LIN {X 0,Y 469.971,Z 691.931,A -85,B 0,C 180,E1 20930.891,E2 20930.891} C_VEL
LIN {X 0,Y 471.709,Z 664.852,A -85,B 0,C 180,E1 20927.125,E2 20927.125} C_VEL
LIN {X 0,Y 473.117,Z 644.354,A -85,B 0,C 180,E1 20924.22,E2 20924.22} C_VEL
LIN {X 0,Y 468.98,Z 629.083,A -85,B 0,C 180,E1 20921.533,E2 20921.533} C_VEL
LIN {X 0,Y 465.017,Z 616.426,A -85,B 0,C 180,E1 20919.107,E2 20919.107} C_VEL
LIN {X 0,Y 465.008,Z 616.312,A -85,B 0,C 180,E1 20915.42,E2 20915.42} C_VEL
LIN {X 0,Y 465.004,Z 616.306,A -85,B 0,C 180,E1 20911.79,E2 20911.79} C_VEL
LIN {X 0,Y 465.007,Z 616.308,A -85,B 0,C 180,E1 20908.093,E2 20908.093} C_VEL
LIN {X 0,Y 465.007,Z 616.309,A -85,B 0,C 180,E1 20904.384,E2 20904.384} C_VEL
LIN {X 0,Y 465.007,Z 616.309,A -85,B 0,C 180,E1 20900.649,E2 20900.649} C_VEL
LIN {X 0,Y 465.005,Z 616.31,A -85,B 0,C 180,E1 20897.004,E2 20897.004} C_VEL
LIN {X 0,Y 465,Z 616.311,A -85,B 0,C 180,E1 20893.302,E2 20893.302} C_VEL
LIN {X 0,Y 465.008,Z 616.3,A -85,B 0,C 180,E1 20889.655,E2 20889.655} C_VEL
LIN {X 0,Y 465.009,Z 616.303,A -85,B 0,C 180,E1 20886.048,E2 20886.048} C_VEL
LIN {X 0,Y 465.002,Z 616.308,A -85,B 0,C 180,E1 20882.342,E2 20882.342} C_VEL
LIN {X 0,Y 464.997,Z 616.312,A -85,B 0,C 180,E1 20878.645,E2 20878.645} C_VEL
LIN {X 0,Y 465.008,Z 616.299,A -85,B 0,C 180,E1 20874.943,E2 20874.943} C_VEL
LIN {X 0,Y 465.01,Z 616.3,A -85,B 0,C 180,E1 20871.344,E2 20871.344} C_VEL
LIN {X 0,Y 465,Z 616.307,A -85,B 0,C 180,E1 20867.709,E2 20867.709} C_VEL
LIN {X 0,Y 464.992,Z 616.314,A -85,B 0,C 180,E1 20864.024,E2 20864.024} C_VEL
LIN {X 0,Y 465.01,Z 616.302,A -85,B 0,C 180,E1 20860.353,E2 20860.353} C_VEL
LIN {X 0,Y 465.01,Z 616.299,A -85,B 0,C 180,E1 20856.654,E2 20856.654} C_VEL
LIN {X 0,Y 465,Z 616.302,A -85,B 0,C 180,E1 20853.019,E2 20853.019} C_VEL
LIN {X 0,Y 464.988,Z 616.304,A -85,B 0,C 180,E1 20849.362,E2 20849.362} C_VEL
LIN {X 0,Y 465.009,Z 616.305,A -85,B 0,C 180,E1 20845.712,E2 20845.712} C_VEL
LIN {X 0,Y 465.014,Z 616.304,A -85,B 0,C 180,E1 20842.052,E2 20842.052} C_VEL
LIN {X 0,Y 464.994,Z 616.31,A -85,B 0,C 180,E1 20838.442,E2 20838.442} C_VEL
LIN {X 0,Y 464.987,Z 616.314,A -85,B 0,C 180,E1 20834.798,E2 20834.798} C_VEL
LIN {X 0,Y 465.018,Z 616.309,A -85,B 0,C 180,E1 20831.143,E2 20831.143} C_VEL
LIN {X 0,Y 465.05,Z 616.559,A -85,B 0,C 180,E1 20829.524,E2 20829.524} C_VEL
LIN {X 0,Y 470.586,Z 631.403,A -85,B 0,C 180,E1 20827.379,E2 20827.379} C_VEL
LIN {X 0,Y 477.306,Z 651.198,A -85,B 0,C 180,E1 20824.859,E2 20824.859} C_VEL
LIN {X 0,Y 474.522,Z 692.791,A -85,B 0,C 180,E1 20821.157,E2 20821.157} C_VEL
LIN {X 0,Y 473.708,Z 708.918,A -85,B 0,C 180,E1 20819.787,E2 20819.787} C_VEL
LIN {X 0,Y 476.659,Z 731.259,A -85,B 0,C 180,E1 20819.245,E2 20819.245} C_VEL
LIN {X 0,Y 474.227,Z 923.8,A -85,B 0,C 180,E1 20816.242,E2 20816.242} C_VEL
LIN {X 0,Y 473.509,Z 943.256,A -85,B 0,C 180,E1 20815.721,E2 20815.721} C_VEL
LIN {X 0,Y 472.588,Z 962.087,A -85,B 0,C 180,E1 20814.99,E2 20814.99} C_VEL
LIN {X 0,Y 471.547,Z 979.642,A -85,B 0,C 180,E1 20814.09,E2 20814.09} C_VEL
LIN {X 0,Y 470.395,Z 997.145,A -85,B 0,C 180,E1 20812.957,E2 20812.957} C_VEL
LIN {X 0,Y 469.201,Z 1013.781,A -85,B 0,C 180,E1 20811.633,E2 20811.633} C_VEL
LIN {X 0,Y 468.041,Z 1029.511,A -85,B 0,C 180,E1 20810.117,E2 20810.117} C_VEL
LIN {X 0,Y 466.991,Z 1043.8,A -85,B 0,C 180,E1 20808.47,E2 20808.47} C_VEL
LIN {X 0,Y 466.038,Z 1057.494,A -85,B 0,C 180,E1 20806.579,E2 20806.579} C_VEL
LIN {X 0,Y 465.315,Z 1068.946,A -85,B 0,C 180,E1 20804.688,E2 20804.688} C_VEL
LIN {X 0,Y 464.744,Z 1079.076,A -85,B 0,C 180,E1 20802.676,E2 20802.676} C_VEL
LIN {X 0,Y 464.358,Z 1087.812,A -85,B 0,C 180,E1 20800.546,E2 20800.546} C_VEL
LIN {X 0,Y 464.099,Z 1095.056,A -85,B 0,C 180,E1 20798.299,E2 20798.299} C_VEL
LIN {X 0,Y 463.962,Z 1100.677,A -85,B 0,C 180,E1 20795.937,E2 20795.937} C_VEL
LIN {X 0,Y 463.915,Z 1104.2,A -85,B 0,C 180,E1 20793.707,E2 20793.707} C_VEL
LIN {X 0,Y 463.911,Z 1106.031,A -85,B 0,C 180,E1 20791.482,E2 20791.482} C_VEL
LIN {X 0,Y 463.912,Z 1106.28,A -85,B 0,C 180,E1 20789.259,E2 20789.259} C_VEL
LIN {X 0,Y 463.911,Z 1104.962,A -85,B 0,C 180,E1 20787.035,E2 20787.035} C_VEL
LIN {X 0,Y 463.937,Z 1102.003,A -85,B 0,C 180,E1 20784.806,E2 20784.806} C_VEL
LIN {X 0,Y 464.031,Z 1097.327,A -85,B 0,C 180,E1 20782.571,E2 20782.571} C_VEL
LIN {X 0,Y 464.235,Z 1090.845,A -85,B 0,C 180,E1 20780.328,E2 20780.328} C_VEL
LIN {X 0,Y 464.56,Z 1082.932,A -85,B 0,C 180,E1 20778.201,E2 20778.201} C_VEL
LIN {X 0,Y 465.072,Z 1073.039,A -85,B 0,C 180,E1 20776.067,E2 20776.067} C_VEL
LIN {X 0,Y 465.772,Z 1061.653,A -85,B 0,C 180,E1 20774.051,E2 20774.051} C_VEL
LIN {X 0,Y 466.645,Z 1048.784,A -85,B 0,C 180,E1 20772.157,E2 20772.157} C_VEL
LIN {X 0,Y 467.708,Z 1034.369,A -85,B 0,C 180,E1 20770.389,E2 20770.389} C_VEL
LIN {X 0,Y 468.856,Z 1018.933,A -85,B 0,C 180,E1 20768.809,E2 20768.809} C_VEL
LIN {X 0,Y 470.058,Z 1002.565,A -85,B 0,C 180,E1 20767.422,E2 20767.422} C_VEL
LIN {X 0,Y 471.25,Z 985.312,A -85,B 0,C 180,E1 20766.226,E2 20766.226} C_VEL
LIN {X 0,Y 472.364,Z 967.12,A -85,B 0,C 180,E1 20765.221,E2 20765.221} C_VEL
LIN {X 0,Y 473.338,Z 948.404,A -85,B 0,C 180,E1 20764.433,E2 20764.433} C_VEL
LIN {X 0,Y 474.13,Z 929.225,A -85,B 0,C 180,E1 20763.861,E2 20763.861} C_VEL
LIN {X 0,Y 474.605,Z 906.118,A -85,B 0,C 180,E1 20763.436,E2 20763.436} C_VEL
LIN {X 0,Y 476.595,Z 728.668,A -85,B 0,C 180,E1 20760.68,E2 20760.68} C_VEL
LIN {X 0,Y 473.739,Z 708.363,A -85,B 0,C 180,E1 20760.163,E2 20760.163} C_VEL
LIN {X 0,Y 476.269,Z 665.707,A -85,B 0,C 180,E1 20756.454,E2 20756.454} C_VEL
LIN {X 0,Y 477.119,Z 650.714,A -85,B 0,C 180,E1 20755.103,E2 20755.103} C_VEL
LIN {X 0,Y 469.453,Z 628.767,A -85,B 0,C 180,E1 20752.401,E2 20752.401} C_VEL
LIN {X 0,Y 465.04,Z 616.516,A -85,B 0,C 180,E1 20750.749,E2 20750.749} C_VEL
LIN {X 0,Y 465.004,Z 616.313,A -85,B 0,C 180,E1 20747.157,E2 20747.157} C_VEL
LIN {X 0,Y 465,Z 616.308,A -85,B 0,C 180,E1 20743.478,E2 20743.478} C_VEL
LIN {X 0,Y 465.016,Z 616.309,A -85,B 0,C 180,E1 20739.847,E2 20739.847} C_VEL
LIN {X 0,Y 464.999,Z 616.313,A -85,B 0,C 180,E1 20736.25,E2 20736.25} C_VEL
LIN {X 0,Y 465.008,Z 616.313,A -85,B 0,C 180,E1 20732.517,E2 20732.517} C_VEL
LIN {X 0,Y 465.014,Z 616.311,A -85,B 0,C 180,E1 20728.792,E2 20728.792} C_VEL
LIN {X 0,Y 465.012,Z 616.31,A -85,B 0,C 180,E1 20725.061,E2 20725.061} C_VEL
LIN {X 0,Y 464.987,Z 616.312,A -85,B 0,C 180,E1 20721.395,E2 20721.395} C_VEL
LIN {X 0,Y 464.98,Z 616.317,A -85,B 0,C 180,E1 20717.649,E2 20717.649} C_VEL
LIN {X 0,Y 465.006,Z 616.315,A -85,B 0,C 180,E1 20714.062,E2 20714.062} C_VEL
LIN {X 0,Y 465.01,Z 616.312,A -85,B 0,C 180,E1 20710.405,E2 20710.405} C_VEL
LIN {X 0,Y 465.002,Z 616.567,A -85,B 0,C 180,E1 20709.311,E2 20709.311} C_VEL
LIN {X 0,Y 469.677,Z 632.432,A -85,B 0,C 180,E1 20707.215,E2 20707.215} C_VEL
LIN {X 0,Y 471.206,Z 640.102,A -85,B 0,C 180,E1 20706.274,E2 20706.274} C_VEL
LIN {X 0,Y 471.027,Z 671.519,A -85,B 0,C 180,E1 20702.737,E2 20702.737} C_VEL
LIN {X 0,Y 470.651,Z 698.884,A -85,B 0,C 180,E1 20699.574,E2 20699.574} C_VEL
LIN {X 0,Y 470.561,Z 708.868,A -85,B 0,C 180,E1 20698.432,E2 20698.432} C_VEL
LIN {X 0,Y 471.035,Z 713.013,A -85,B 0,C 180,E1 20698.329,E2 20698.329} C_VEL
LIN {X 0,Y 469.379,Z 847.569,A -85,B 0,C 180,E1 20696.041,E2 20696.041} C_VEL
LIN {X 0,Y 469.234,Z 863.454,A -85,B 0,C 180,E1 20695.554,E2 20695.554} C_VEL
LIN {X 0,Y 468.89,Z 879.333,A -85,B 0,C 180,E1 20694.826,E2 20694.826} C_VEL
LIN {X 0,Y 468.431,Z 893.617,A -85,B 0,C 180,E1 20693.935,E2 20693.935} C_VEL
LIN {X 0,Y 467.831,Z 908.134,A -85,B 0,C 180,E1 20692.756,E2 20692.756} C_VEL
LIN {X 0,Y 467.229,Z 920.197,A -85,B 0,C 180,E1 20691.508,E2 20691.508} C_VEL
LIN {X 0,Y 466.592,Z 931.837,A -85,B 0,C 180,E1 20690.004,E2 20690.004} C_VEL
LIN {X 0,Y 466.055,Z 941.162,A -85,B 0,C 180,E1 20688.491,E2 20688.491} C_VEL
LIN {X 0,Y 465.573,Z 949.787,A -85,B 0,C 180,E1 20686.715,E2 20686.715} C_VEL
LIN {X 0,Y 465.223,Z 956.426,A -85,B 0,C 180,E1 20684.926,E2 20684.926} C_VEL
LIN {X 0,Y 464.953,Z 961.615,A -85,B 0,C 180,E1 20682.994,E2 20682.994} C_VEL
LIN {X 0,Y 464.788,Z 965.016,A -85,B 0,C 180,E1 20681.044,E2 20681.044} C_VEL
LIN {X 0,Y 464.699,Z 966.73,A -85,B 0,C 180,E1 20678.941,E2 20678.941} C_VEL
LIN {X 0,Y 464.68,Z 966.571,A -85,B 0,C 180,E1 20676.945,E2 20676.945} C_VEL
LIN {X 0,Y 464.716,Z 964.62,A -85,B 0,C 180,E1 20674.921,E2 20674.921} C_VEL
LIN {X 0,Y 464.835,Z 960.927,A -85,B 0,C 180,E1 20672.939,E2 20672.939} C_VEL
LIN {X 0,Y 465.064,Z 955.222,A -85,B 0,C 180,E1 20670.929,E2 20670.929} C_VEL
LIN {X 0,Y 465.382,Z 948.093,A -85,B 0,C 180,E1 20669.103,E2 20669.103} C_VEL
LIN {X 0,Y 465.852,Z 938.867,A -85,B 0,C 180,E1 20667.284,E2 20667.284} C_VEL
LIN {X 0,Y 466.395,Z 928.44,A -85,B 0,C 180,E1 20665.679,E2 20665.679} C_VEL
LIN {X 0,Y 467.011,Z 916.752,A -85,B 0,C 180,E1 20664.233,E2 20664.233} C_VEL
LIN {X 0,Y 467.592,Z 904.339,A -85,B 0,C 180,E1 20663.008,E2 20663.008} C_VEL
LIN {X 0,Y 468.199,Z 890.125,A -85,B 0,C 180,E1 20661.89,E2 20661.89} C_VEL
LIN {X 0,Y 468.692,Z 875.343,A -85,B 0,C 180,E1 20660.999,E2 20660.999} C_VEL
LIN {X 0,Y 469.089,Z 858.993,A -85,B 0,C 180,E1 20660.276,E2 20660.276} C_VEL
LIN {X 0,Y 469.274,Z 842.347,A -85,B 0,C 180,E1 20659.8,E2 20659.8} C_VEL
LIN {X 0,Y 469.47,Z 814.945,A -85,B 0,C 180,E1 20659.337,E2 20659.337} C_VEL
LIN {X 0,Y 468.618,Z 807.338,A -85,B 0,C 180,E1 20659.179,E2 20659.179} C_VEL
LIN {X 0,Y 462.907,Z 787.393,A -85,B 0,C 180,E1 20658.614,E2 20658.614} C_VEL
LIN {X 0,Y 462.253,Z 780.859,A -85,B 0,C 180,E1 20658.475,E2 20658.475} C_VEL
LIN {X 0,Y 463.052,Z 710.901,A -85,B 0,C 180,E1 20657.29,E2 20657.29} C_VEL
LIN {X 0,Y 461.82,Z 704.156,A -85,B 0,C 180,E1 20657.082,E2 20657.082} C_VEL
LIN {X 0,Y 462.508,Z 674.571,A -85,B 0,C 180,E1 20653.505,E2 20653.505} C_VEL
LIN {X 0,Y 463.139,Z 645.733,A -85,B 0,C 180,E1 20650.042,E2 20650.042} C_VEL
LIN {X 0,Y 463.021,Z 640.199,A -85,B 0,C 180,E1 20649.369,E2 20649.369} C_VEL
LIN {X 0,Y 458.266,Z 621.938,A -85,B 0,C 180,E1 20646.871,E2 20646.871} C_VEL
LIN {X 0,Y 457.05,Z 617.433,A -85,B 0,C 180,E1 20646.172,E2 20646.172} C_VEL
LIN {X 0,Y 457.013,Z 617.3,A -85,B 0,C 180,E1 20642.562,E2 20642.562} C_VEL
LIN {X 0,Y 457.034,Z 617.301,A -85,B 0,C 180,E1 20638.914,E2 20638.914} C_VEL
LIN {X 0,Y 457.066,Z 617.275,A -85,B 0,C 180,E1 20635.382,E2 20635.382} C_VEL
LIN {X 0,Y 457.03,Z 617.307,A -85,B 0,C 180,E1 20631.834,E2 20631.834} C_VEL
LIN {X 0,Y 457.025,Z 617.305,A -85,B 0,C 180,E1 20628.099,E2 20628.099} C_VEL
LIN {X 0,Y 457.076,Z 617.575,A -85,B 0,C 180,E1 20626.304,E2 20626.304} C_VEL
LIN {X 0,Y 462.186,Z 635.495,A -85,B 0,C 180,E1 20623.219,E2 20623.219} C_VEL
LIN {X 0,Y 464.604,Z 645.672,A -85,B 0,C 180,E1 20621.546,E2 20621.546} C_VEL
LIN {X 0,Y 462.93,Z 672.491,A -85,B 0,C 180,E1 20617.821,E2 20617.821} C_VEL
LIN {X 0,Y 461.677,Z 693.969,A -85,B 0,C 180,E1 20614.877,E2 20614.877} C_VEL
LIN {X 0,Y 462.728,Z 699.529,A -85,B 0,C 180,E1 20614.676,E2 20614.676} C_VEL
LIN {X 0,Y 465.629,Z 714.224,A -85,B 0,C 180,E1 20614.278,E2 20614.278} C_VEL
LIN {X 0,Y 463.988,Z 841.192,A -85,B 0,C 180,E1 20612.219,E2 20612.219} C_VEL
LIN {X 0,Y 463.588,Z 858.183,A -85,B 0,C 180,E1 20611.7,E2 20611.7} C_VEL
LIN {X 0,Y 463.006,Z 873.88,A -85,B 0,C 180,E1 20610.99,E2 20610.99} C_VEL
LIN {X 0,Y 462.224,Z 888.912,A -85,B 0,C 180,E1 20610.062,E2 20610.062} C_VEL
LIN {X 0,Y 461.349,Z 903.005,A -85,B 0,C 180,E1 20608.945,E2 20608.945} C_VEL
LIN {X 0,Y 460.452,Z 916.069,A -85,B 0,C 180,E1 20607.636,E2 20607.636} C_VEL
LIN {X 0,Y 459.546,Z 928.054,A -85,B 0,C 180,E1 20606.133,E2 20606.133} C_VEL
LIN {X 0,Y 458.728,Z 938.568,A -85,B 0,C 180,E1 20604.497,E2 20604.497} C_VEL
LIN {X 0,Y 458.034,Z 947.543,A -85,B 0,C 180,E1 20602.727,E2 20602.727} C_VEL
LIN {X 0,Y 457.499,Z 955.088,A -85,B 0,C 180,E1 20600.82,E2 20600.82} C_VEL
LIN {X 0,Y 457.148,Z 960.753,A -85,B 0,C 180,E1 20598.903,E2 20598.903} C_VEL
LIN {X 0,Y 456.907,Z 964.939,A -85,B 0,C 180,E1 20596.845,E2 20596.845} C_VEL
LIN {X 0,Y 456.798,Z 967.407,A -85,B 0,C 180,E1 20594.772,E2 20594.772} C_VEL
LIN {X 0,Y 456.776,Z 968.111,A -85,B 0,C 180,E1 20592.628,E2 20592.628} C_VEL
LIN {X 0,Y 456.858,Z 967.01,A -85,B 0,C 180,E1 20590.437,E2 20590.437} C_VEL
LIN {X 0,Y 457.048,Z 964.236,A -85,B 0,C 180,E1 20588.397,E2 20588.397} C_VEL
LIN {X 0,Y 457.376,Z 959.482,A -85,B 0,C 180,E1 20586.282,E2 20586.282} C_VEL
LIN {X 0,Y 457.84,Z 953.455,A -85,B 0,C 180,E1 20584.38,E2 20584.38} C_VEL
LIN {X 0,Y 458.504,Z 945.336,A -85,B 0,C 180,E1 20582.464,E2 20582.464} C_VEL
LIN {X 0,Y 459.356,Z 935.665,A -85,B 0,C 180,E1 20580.676,E2 20580.676} C_VEL
LIN {X 0,Y 460.276,Z 924.892,A -85,B 0,C 180,E1 20579.1,E2 20579.1} C_VEL
LIN {X 0,Y 461.287,Z 912.392,A -85,B 0,C 180,E1 20577.63,E2 20577.63} C_VEL
LIN {X 0,Y 462.277,Z 899.06,A -85,B 0,C 180,E1 20576.379,E2 20576.379} C_VEL
LIN {X 0,Y 463.157,Z 884.94,A -85,B 0,C 180,E1 20575.336,E2 20575.336} C_VEL
LIN {X 0,Y 463.958,Z 869.563,A -85,B 0,C 180,E1 20574.462,E2 20574.462} C_VEL
LIN {X 0,Y 464.524,Z 853.564,A -85,B 0,C 180,E1 20573.809,E2 20573.809} C_VEL
LIN {X 0,Y 464.857,Z 836.203,A -85,B 0,C 180,E1 20573.357,E2 20573.357} C_VEL
LIN {X 0,Y 466.5,Z 712.866,A -85,B 0,C 180,E1 20571.326,E2 20571.326} C_VEL
LIN {X 0,Y 462.486,Z 694.526,A -85,B 0,C 180,E1 20570.712,E2 20570.712} C_VEL
LIN {X 0,Y 464.196,Z 668.574,A -85,B 0,C 180,E1 20567.084,E2 20567.084} C_VEL
LIN {X 0,Y 465.809,Z 647.249,A -85,B 0,C 180,E1 20564.022,E2 20564.022} C_VEL
LIN {X 0,Y 461.675,Z 631.95,A -85,B 0,C 180,E1 20561.279,E2 20561.279} C_VEL
LIN {X 0,Y 457.082,Z 617.422,A -85,B 0,C 180,E1 20558.432,E2 20558.432} C_VEL
LIN {X 0,Y 457.068,Z 617.304,A -85,B 0,C 180,E1 20554.817,E2 20554.817} C_VEL
LIN {X 0,Y 457.067,Z 617.293,A -85,B 0,C 180,E1 20551.082,E2 20551.082} C_VEL
LIN {X 0,Y 457.071,Z 617.3,A -85,B 0,C 180,E1 20547.36,E2 20547.36} C_VEL
LIN {X 0,Y 457.061,Z 617.3,A -85,B 0,C 180,E1 20543.599,E2 20543.599} C_VEL
LIN {X 0,Y 457.072,Z 617.301,A -85,B 0,C 180,E1 20539.954,E2 20539.954} C_VEL
LIN {X 0,Y 457.068,Z 617.302,A -85,B 0,C 180,E1 20536.192,E2 20536.192} C_VEL
LIN {X 0,Y 457.073,Z 617.297,A -85,B 0,C 180,E1 20532.508,E2 20532.508} C_VEL
LIN {X 0,Y 457.06,Z 617.299,A -85,B 0,C 180,E1 20528.809,E2 20528.809} C_VEL
LIN {X 0,Y 457.063,Z 617.29,A -85,B 0,C 180,E1 20525.146,E2 20525.146} C_VEL
LIN {X 0,Y 457.07,Z 617.29,A -85,B 0,C 180,E1 20521.396,E2 20521.396} C_VEL
LIN {X 0,Y 457.071,Z 617.298,A -85,B 0,C 180,E1 20517.618,E2 20517.618} C_VEL
LIN {X 0,Y 457.069,Z 617.295,A -85,B 0,C 180,E1 20513.847,E2 20513.847} C_VEL
LIN {X 0,Y 457.054,Z 617.291,A -85,B 0,C 180,E1 20510.176,E2 20510.176} C_VEL
LIN {X 0,Y 457.068,Z 617.287,A -85,B 0,C 180,E1 20506.464,E2 20506.464} C_VEL
LIN {X 0,Y 457.072,Z 617.301,A -85,B 0,C 180,E1 20502.824,E2 20502.824} C_VEL
LIN {X 0,Y 457.074,Z 617.297,A -85,B 0,C 180,E1 20499.078,E2 20499.078} C_VEL
LIN {X 0,Y 457.052,Z 617.301,A -85,B 0,C 180,E1 20495.44,E2 20495.44} C_VEL
LIN {X 0,Y 457.058,Z 617.298,A -85,B 0,C 180,E1 20491.66,E2 20491.66} C_VEL
LIN {X 0,Y 457.075,Z 617.291,A -85,B 0,C 180,E1 20488.037,E2 20488.037} C_VEL
LIN {X 0,Y 457.072,Z 617.295,A -85,B 0,C 180,E1 20484.263,E2 20484.263} C_VEL
LIN {X 0,Y 457.057,Z 617.302,A -85,B 0,C 180,E1 20480.554,E2 20480.554} C_VEL
LIN {X 0,Y 457.05,Z 617.298,A -85,B 0,C 180,E1 20476.942,E2 20476.942} C_VEL
LIN {X 0,Y 457.07,Z 617.299,A -85,B 0,C 180,E1 20473.212,E2 20473.212} C_VEL
LIN {X 0,Y 457.089,Z 617.569,A -85,B 0,C 180,E1 20470.21,E2 20470.21} C_VEL
LIN {X 0,Y 463.034,Z 633.107,A -85,B 0,C 180,E1 20467.885,E2 20467.885} C_VEL
LIN {X 0,Y 469.513,Z 652.343,A -85,B 0,C 180,E1 20465.351,E2 20465.351} C_VEL
LIN {X 0,Y 470.025,Z 654.933,A -85,B 0,C 180,E1 20465.054,E2 20465.054} C_VEL
LIN {X 0,Y 466.972,Z 696.448,A -85,B 0,C 180,E1 20461.287,E2 20461.287} C_VEL
LIN {X 0,Y 466.347,Z 708.899,A -85,B 0,C 180,E1 20460.227,E2 20460.227} C_VEL
LIN {X 0,Y 469.41,Z 732.338,A -85,B 0,C 180,E1 20459.643,E2 20459.643} C_VEL
LIN {X 0,Y 466.804,Z 923.096,A -85,B 0,C 180,E1 20456.615,E2 20456.615} C_VEL
LIN {X 0,Y 466.041,Z 942.504,A -85,B 0,C 180,E1 20456.087,E2 20456.087} C_VEL
LIN {X 0,Y 465.075,Z 960.929,A -85,B 0,C 180,E1 20455.364,E2 20455.364} C_VEL
LIN {X 0,Y 463.962,Z 978.681,A -85,B 0,C 180,E1 20454.441,E2 20454.441} C_VEL
LIN {X 0,Y 462.738,Z 996.18,A -85,B 0,C 180,E1 20453.292,E2 20453.292} C_VEL
LIN {X 0,Y 461.504,Z 1012.374,A -85,B 0,C 180,E1 20451.987,E2 20451.987} C_VEL
LIN {X 0,Y 460.236,Z 1028.527,A -85,B 0,C 180,E1 20450.407,E2 20450.407} C_VEL
LIN {X 0,Y 459.091,Z 1043.283,A -85,B 0,C 180,E1 20448.668,E2 20448.668} C_VEL
LIN {X 0,Y 458.151,Z 1056.07,A -85,B 0,C 180,E1 20446.873,E2 20446.873} C_VEL
LIN {X 0,Y 457.389,Z 1067.644,A -85,B 0,C 180,E1 20444.936,E2 20444.936} C_VEL
LIN {X 0,Y 456.772,Z 1078.303,A -85,B 0,C 180,E1 20442.772,E2 20442.772} C_VEL
LIN {X 0,Y 456.391,Z 1086.967,A -85,B 0,C 180,E1 20440.604,E2 20440.604} C_VEL
LIN {X 0,Y 456.143,Z 1094.138,A -85,B 0,C 180,E1 20438.318,E2 20438.318} C_VEL
LIN {X 0,Y 456.027,Z 1099.454,A -85,B 0,C 180,E1 20436.041,E2 20436.041} C_VEL
LIN {X 0,Y 455.99,Z 1103.164,A -85,B 0,C 180,E1 20433.646,E2 20433.646} C_VEL
LIN {X 0,Y 455.988,Z 1105.024,A -85,B 0,C 180,E1 20431.256,E2 20431.256} C_VEL
LIN {X 0,Y 455.989,Z 1105.094,A -85,B 0,C 180,E1 20428.995,E2 20428.995} C_VEL
LIN {X 0,Y 455.991,Z 1103.549,A -85,B 0,C 180,E1 20426.731,E2 20426.731} C_VEL
LIN {X 0,Y 456.011,Z 1100.363,A -85,B 0,C 180,E1 20424.463,E2 20424.463} C_VEL
LIN {X 0,Y 456.098,Z 1095.465,A -85,B 0,C 180,E1 20422.188,E2 20422.188} C_VEL
LIN {X 0,Y 456.316,Z 1088.747,A -85,B 0,C 180,E1 20419.904,E2 20419.904} C_VEL
LIN {X 0,Y 456.691,Z 1080.031,A -85,B 0,C 180,E1 20417.61,E2 20417.61} C_VEL
LIN {X 0,Y 457.269,Z 1069.724,A -85,B 0,C 180,E1 20415.436,E2 20415.436} C_VEL
LIN {X 0,Y 458.046,Z 1057.872,A -85,B 0,C 180,E1 20413.384,E2 20413.384} C_VEL
LIN {X 0,Y 459.031,Z 1044.468,A -85,B 0,C 180,E1 20411.457,E2 20411.457} C_VEL
LIN {X 0,Y 460.163,Z 1029.996,A -85,B 0,C 180,E1 20409.722,E2 20409.722} C_VEL
LIN {X 0,Y 461.382,Z 1014.588,A -85,B 0,C 180,E1 20408.182,E2 20408.182} C_VEL
LIN {X 0,Y 462.673,Z 997.9,A -85,B 0,C 180,E1 20406.803,E2 20406.803} C_VEL
LIN {X 0,Y 463.928,Z 980.322,A -85,B 0,C 180,E1 20405.624,E2 20405.624} C_VEL
LIN {X 0,Y 465.081,Z 962.329,A -85,B 0,C 180,E1 20404.67,E2 20404.67} C_VEL
LIN {X 0,Y 466.083,Z 943.437,A -85,B 0,C 180,E1 20403.914,E2 20403.914} C_VEL
LIN {X 0,Y 466.852,Z 924.232,A -85,B 0,C 180,E1 20403.383,E2 20403.383} C_VEL
LIN {X 0,Y 467.504,Z 879.708,A -85,B 0,C 180,E1 20402.654,E2 20402.654} C_VEL
LIN {X 0,Y 469.314,Z 729.656,A -85,B 0,C 180,E1 20400.284,E2 20400.284} C_VEL
LIN {X 0,Y 466.332,Z 708.168,A -85,B 0,C 180,E1 20399.726,E2 20399.726} C_VEL
LIN {X 0,Y 468.914,Z 668.19,A -85,B 0,C 180,E1 20396.184,E2 20396.184} C_VEL
LIN {X 0,Y 469.89,Z 653.695,A -85,B 0,C 180,E1 20394.869,E2 20394.869} C_VEL
LIN {X 0,Y 462.162,Z 631.537,A -85,B 0,C 180,E1 20392.09,E2 20392.09} C_VEL
LIN {X 0,Y 457.103,Z 617.506,A -85,B 0,C 180,E1 20390.174,E2 20390.174} C_VEL
LIN {X 0,Y 457.07,Z 617.299,A -85,B 0,C 180,E1 20386.574,E2 20386.574} C_VEL
LIN {X 0,Y 457.071,Z 617.302,A -85,B 0,C 180,E1 20382.869,E2 20382.869} C_VEL
LIN {X 0,Y 457.064,Z 617.299,A -85,B 0,C 180,E1 20379.213,E2 20379.213} C_VEL
LIN {X 0,Y 457.071,Z 617.299,A -85,B 0,C 180,E1 20375.534,E2 20375.534} C_VEL
LIN {X 0,Y 457.059,Z 617.3,A -85,B 0,C 180,E1 20371.817,E2 20371.817} C_VEL
LIN {X 0,Y 457.055,Z 617.301,A -85,B 0,C 180,E1 20368.056,E2 20368.056} C_VEL
LIN {X 0,Y 457.072,Z 617.302,A -85,B 0,C 180,E1 20364.421,E2 20364.421} C_VEL
LIN {X 0,Y 457.08,Z 617.3,A -85,B 0,C 180,E1 20360.755,E2 20360.755} C_VEL
LIN {X 0,Y 457.051,Z 617.303,A -85,B 0,C 180,E1 20357.046,E2 20357.046} C_VEL
LIN {X 0,Y 457.032,Z 617.307,A -85,B 0,C 180,E1 20353.409,E2 20353.409} C_VEL
LIN {X 0,Y 457.08,Z 617.502,A -85,B 0,C 180,E1 20349.824,E2 20349.824} C_VEL
LIN {X 0,Y 461.8,Z 633.15,A -85,B 0,C 180,E1 20347.714,E2 20347.714} C_VEL
LIN {X 0,Y 463.853,Z 642.219,A -85,B 0,C 180,E1 20346.56,E2 20346.56} C_VEL
LIN {X 0,Y 463.692,Z 670.814,A -85,B 0,C 180,E1 20343.337,E2 20343.337} C_VEL
LIN {X 0,Y 463.318,Z 697.587,A -85,B 0,C 180,E1 20340.247,E2 20340.247} C_VEL
LIN {X 0,Y 463.157,Z 710.122,A -85,B 0,C 180,E1 20338.794,E2 20338.794} C_VEL
LIN {X 0,Y 463.618,Z 714.293,A -85,B 0,C 180,E1 20338.683,E2 20338.683} C_VEL
LIN {X 0,Y 461.808,Z 848.914,A -85,B 0,C 180,E1 20336.334,E2 20336.334} C_VEL
LIN {X 0,Y 461.662,Z 864.785,A -85,B 0,C 180,E1 20335.839,E2 20335.839} C_VEL
LIN {X 0,Y 461.297,Z 880.865,A -85,B 0,C 180,E1 20335.088,E2 20335.088} C_VEL
LIN {X 0,Y 460.825,Z 894.814,A -85,B 0,C 180,E1 20334.204,E2 20334.204} C_VEL
LIN {X 0,Y 460.188,Z 909.281,A -85,B 0,C 180,E1 20333.011,E2 20333.011} C_VEL
LIN {X 0,Y 459.547,Z 921.376,A -85,B 0,C 180,E1 20331.744,E2 20331.744} C_VEL
LIN {X 0,Y 458.862,Z 933.026,A -85,B 0,C 180,E1 20330.214,E2 20330.214} C_VEL
LIN {X 0,Y 458.285,Z 942.378,A -85,B 0,C 180,E1 20328.676,E2 20328.676} C_VEL
LIN {X 0,Y 457.761,Z 951.019,A -85,B 0,C 180,E1 20326.87,E2 20326.87} C_VEL
LIN {X 0,Y 457.378,Z 957.67,A -85,B 0,C 180,E1 20325.051,E2 20325.051} C_VEL
LIN {X 0,Y 457.079,Z 962.86,A -85,B 0,C 180,E1 20323.086,E2 20323.086} C_VEL
LIN {X 0,Y 456.896,Z 966.256,A -85,B 0,C 180,E1 20321.102,E2 20321.102} C_VEL
LIN {X 0,Y 456.795,Z 967.956,A -85,B 0,C 180,E1 20318.963,E2 20318.963} C_VEL
LIN {X 0,Y 456.771,Z 967.772,A -85,B 0,C 180,E1 20316.932,E2 20316.932} C_VEL
LIN {X 0,Y 456.811,Z 965.797,A -85,B 0,C 180,E1 20314.873,E2 20314.873} C_VEL
LIN {X 0,Y 456.936,Z 962.23,A -85,B 0,C 180,E1 20312.926,E2 20312.926} C_VEL
LIN {X 0,Y 457.167,Z 956.773,A -85,B 0,C 180,E1 20310.952,E2 20310.952} C_VEL
LIN {X 0,Y 457.505,Z 949.772,A -85,B 0,C 180,E1 20309.097,E2 20309.097} C_VEL
LIN {X 0,Y 457.998,Z 940.49,A -85,B 0,C 180,E1 20307.22,E2 20307.22} C_VEL
LIN {X 0,Y 458.562,Z 930.386,A -85,B 0,C 180,E1 20305.616,E2 20305.616} C_VEL
LIN {X 0,Y 459.226,Z 918.371,A -85,B 0,C 180,E1 20304.091,E2 20304.091} C_VEL
LIN {X 0,Y 459.859,Z 905.698,A -85,B 0,C 180,E1 20302.81,E2 20302.81} C_VEL
LIN {X 0,Y 460.496,Z 891.477,A -85,B 0,C 180,E1 20301.671,E2 20301.671} C_VEL
LIN {X 0,Y 461.003,Z 877.107,A -85,B 0,C 180,E1 20300.782,E2 20300.782} C_VEL
LIN {X 0,Y 461.425,Z 860.556,A -85,B 0,C 180,E1 20300.03,E2 20300.03} C_VEL
LIN {X 0,Y 461.621,Z 844.321,A -85,B 0,C 180,E1 20299.547,E2 20299.547} C_VEL
LIN {X 0,Y 462.253,Z 780.859,A -85,B 0,C 180,E1 20298.475,E2 20298.475} C_VEL
LIN {X 0,Y 461.387,Z 773.257,A -85,B 0,C 180,E1 20298.308,E2 20298.308} C_VEL
LIN {X 0,Y 455.788,Z 753.323,A -85,B 0,C 180,E1 20297.713,E2 20297.713} C_VEL
LIN {X 0,Y 455.191,Z 746.791,A -85,B 0,C 180,E1 20297.57,E2 20297.57} C_VEL
LIN {X 0,Y 455.503,Z 711.927,A -85,B 0,C 180,E1 20296.961,E2 20296.961} C_VEL
LIN {X 0,Y 454.281,Z 705.291,A -85,B 0,C 180,E1 20296.763,E2 20296.763} C_VEL
LIN {X 0,Y 454.983,Z 675.907,A -85,B 0,C 180,E1 20293.2,E2 20293.2} C_VEL
LIN {X 0,Y 455.65,Z 646.232,A -85,B 0,C 180,E1 20289.626,E2 20289.626} C_VEL
LIN {X 0,Y 455.354,Z 641.82,A -85,B 0,C 180,E1 20289.065,E2 20289.065} C_VEL
LIN {X 0,Y 450.7,Z 624.223,A -85,B 0,C 180,E1 20286.639,E2 20286.639} C_VEL
LIN {X 0,Y 449.144,Z 618.422,A -85,B 0,C 180,E1 20285.757,E2 20285.757} C_VEL
LIN {X 0,Y 449.087,Z 618.29,A -85,B 0,C 180,E1 20282.149,E2 20282.149} C_VEL
LIN {X 0,Y 449.078,Z 618.291,A -85,B 0,C 180,E1 20278.455,E2 20278.455} C_VEL
LIN {X 0,Y 449.105,Z 618.261,A -85,B 0,C 180,E1 20274.884,E2 20274.884} C_VEL
LIN {X 0,Y 449.133,Z 618.281,A -85,B 0,C 180,E1 20271.277,E2 20271.277} C_VEL
LIN {X 0,Y 449.096,Z 618.295,A -85,B 0,C 180,E1 20267.625,E2 20267.625} C_VEL
LIN {X 0,Y 449.183,Z 618.619,A -85,B 0,C 180,E1 20266.821,E2 20266.821} C_VEL
LIN {X 0,Y 454.388,Z 636.845,A -85,B 0,C 180,E1 20263.618,E2 20263.618} C_VEL
LIN {X 0,Y 457.095,Z 648.083,A -85,B 0,C 180,E1 20261.738,E2 20261.738} C_VEL
LIN {X 0,Y 455.257,Z 675.939,A -85,B 0,C 180,E1 20257.826,E2 20257.826} C_VEL
LIN {X 0,Y 454.161,Z 694.475,A -85,B 0,C 180,E1 20255.274,E2 20255.274} C_VEL
LIN {X 0,Y 458.306,Z 715.459,A -85,B 0,C 180,E1 20254.664,E2 20254.664} C_VEL
LIN {X 0,Y 456.578,Z 841.727,A -85,B 0,C 180,E1 20252.589,E2 20252.589} C_VEL
LIN {X 0,Y 456.162,Z 858.696,A -85,B 0,C 180,E1 20252.065,E2 20252.065} C_VEL
LIN {X 0,Y 455.579,Z 873.732,A -85,B 0,C 180,E1 20251.384,E2 20251.384} C_VEL
LIN {X 0,Y 454.813,Z 888.177,A -85,B 0,C 180,E1 20250.504,E2 20250.504} C_VEL
LIN {X 0,Y 453.872,Z 902.579,A -85,B 0,C 180,E1 20249.369,E2 20249.369} C_VEL
LIN {X 0,Y 452.911,Z 915.968,A -85,B 0,C 180,E1 20248.039,E2 20248.039} C_VEL
LIN {X 0,Y 451.971,Z 927.705,A -85,B 0,C 180,E1 20246.576,E2 20246.576} C_VEL
LIN {X 0,Y 451.069,Z 938.466,A -85,B 0,C 180,E1 20244.913,E2 20244.913} C_VEL
LIN {X 0,Y 450.309,Z 947.742,A -85,B 0,C 180,E1 20243.114,E2 20243.114} C_VEL
LIN {X 0,Y 449.706,Z 955.472,A -85,B 0,C 180,E1 20241.176,E2 20241.176} C_VEL
LIN {X 0,Y 449.303,Z 961.358,A -85,B 0,C 180,E1 20239.227,E2 20239.227} C_VEL
LIN {X 0,Y 449.032,Z 965.749,A -85,B 0,C 180,E1 20237.134,E2 20237.134} C_VEL
LIN {X 0,Y 448.89,Z 968.5,A -85,B 0,C 180,E1 20234.894,E2 20234.894} C_VEL
LIN {X 0,Y 448.865,Z 969.326,A -85,B 0,C 180,E1 20232.767,E2 20232.767} C_VEL
LIN {X 0,Y 448.941,Z 968.412,A -85,B 0,C 180,E1 20230.62,E2 20230.62} C_VEL
LIN {X 0,Y 449.157,Z 965.742,A -85,B 0,C 180,E1 20228.451,E2 20228.451} C_VEL
LIN {X 0,Y 449.482,Z 961.384,A -85,B 0,C 180,E1 20226.397,E2 20226.397} C_VEL
LIN {X 0,Y 450.008,Z 955.126,A -85,B 0,C 180,E1 20224.325,E2 20224.325} C_VEL
LIN {X 0,Y 450.668,Z 947.868,A -85,B 0,C 180,E1 20222.518,E2 20222.518} C_VEL
LIN {X 0,Y 451.541,Z 938.515,A -85,B 0,C 180,E1 20220.701,E2 20220.701} C_VEL
LIN {X 0,Y 452.58,Z 927.557,A -85,B 0,C 180,E1 20219.003,E2 20219.003} C_VEL
LIN {X 0,Y 453.616,Z 915.768,A -85,B 0,C 180,E1 20217.547,E2 20217.547} C_VEL
LIN {X 0,Y 454.715,Z 902.157,A -85,B 0,C 180,E1 20216.199,E2 20216.199} C_VEL
LIN {X 0,Y 455.689,Z 888.274,A -85,B 0,C 180,E1 20215.111,E2 20215.111} C_VEL
LIN {X 0,Y 456.569,Z 872.697,A -85,B 0,C 180,E1 20214.179,E2 20214.179} C_VEL
LIN {X 0,Y 457.234,Z 856.368,A -85,B 0,C 180,E1 20213.463,E2 20213.463} C_VEL
LIN {X 0,Y 457.601,Z 839.674,A -85,B 0,C 180,E1 20212.992,E2 20212.992} C_VEL
LIN {X 0,Y 459.434,Z 714.249,A -85,B 0,C 180,E1 20210.879,E2 20210.879} C_VEL
LIN {X 0,Y 455.128,Z 694.731,A -85,B 0,C 180,E1 20210.207,E2 20210.207} C_VEL
LIN {X 0,Y 456.97,Z 668.697,A -85,B 0,C 180,E1 20206.518,E2 20206.518} C_VEL
LIN {X 0,Y 458.405,Z 649.726,A -85,B 0,C 180,E1 20203.744,E2 20203.744} C_VEL
LIN {X 0,Y 454.336,Z 634.651,A -85,B 0,C 180,E1 20200.982,E2 20200.982} C_VEL
LIN {X 0,Y 449.999,Z 621.089,A -85,B 0,C 180,E1 20198.31,E2 20198.31} C_VEL
LIN {X 0,Y 449.149,Z 618.398,A -85,B 0,C 180,E1 20197.704,E2 20197.704} C_VEL
LIN {X 0,Y 449.126,Z 618.284,A -85,B 0,C 180,E1 20193.972,E2 20193.972} C_VEL
LIN {X 0,Y 449.135,Z 618.291,A -85,B 0,C 180,E1 20190.207,E2 20190.207} C_VEL
LIN {X 0,Y 449.13,Z 618.287,A -85,B 0,C 180,E1 20186.439,E2 20186.439} C_VEL
LIN {X 0,Y 449.128,Z 618.283,A -85,B 0,C 180,E1 20182.653,E2 20182.653} C_VEL
LIN {X 0,Y 449.132,Z 618.279,A -85,B 0,C 180,E1 20178.892,E2 20178.892} C_VEL
LIN {X 0,Y 449.118,Z 618.281,A -85,B 0,C 180,E1 20175.231,E2 20175.231} C_VEL
LIN {X 0,Y 449.129,Z 618.286,A -85,B 0,C 180,E1 20171.558,E2 20171.558} C_VEL
LIN {X 0,Y 449.131,Z 618.289,A -85,B 0,C 180,E1 20167.805,E2 20167.805} C_VEL
LIN {X 0,Y 449.131,Z 618.283,A -85,B 0,C 180,E1 20164.085,E2 20164.085} C_VEL
LIN {X 0,Y 449.118,Z 618.276,A -85,B 0,C 180,E1 20160.383,E2 20160.383} C_VEL
LIN {X 0,Y 449.118,Z 618.277,A -85,B 0,C 180,E1 20156.682,E2 20156.682} C_VEL
LIN {X 0,Y 449.138,Z 618.289,A -85,B 0,C 180,E1 20152.967,E2 20152.967} C_VEL
LIN {X 0,Y 449.131,Z 618.282,A -85,B 0,C 180,E1 20149.222,E2 20149.222} C_VEL
LIN {X 0,Y 449.134,Z 618.275,A -85,B 0,C 180,E1 20145.43,E2 20145.43} C_VEL
LIN {X 0,Y 449.115,Z 618.275,A -85,B 0,C 180,E1 20141.705,E2 20141.705} C_VEL
LIN {X 0,Y 449.119,Z 618.282,A -85,B 0,C 180,E1 20137.899,E2 20137.899} C_VEL
LIN {X 0,Y 449.133,Z 618.288,A -85,B 0,C 180,E1 20134.13,E2 20134.13} C_VEL
LIN {X 0,Y 449.137,Z 618.289,A -85,B 0,C 180,E1 20130.382,E2 20130.382} C_VEL
LIN {X 0,Y 449.131,Z 618.288,A -85,B 0,C 180,E1 20126.597,E2 20126.597} C_VEL
LIN {X 0,Y 449.111,Z 618.288,A -85,B 0,C 180,E1 20122.846,E2 20122.846} C_VEL
LIN {X 0,Y 449.114,Z 618.285,A -85,B 0,C 180,E1 20119.116,E2 20119.116} C_VEL
LIN {X 0,Y 449.135,Z 618.288,A -85,B 0,C 180,E1 20115.429,E2 20115.429} C_VEL
LIN {X 0,Y 449.135,Z 618.284,A -85,B 0,C 180,E1 20111.73,E2 20111.73} C_VEL
LIN {X 0,Y 449.173,Z 618.624,A -85,B 0,C 180,E1 20110.931,E2 20110.931} C_VEL
LIN {X 0,Y 455.468,Z 634.896,A -85,B 0,C 180,E1 20108.4,E2 20108.4} C_VEL
LIN {X 0,Y 461.648,Z 653.19,A -85,B 0,C 180,E1 20105.902,E2 20105.902} C_VEL
LIN {X 0,Y 462.838,Z 657.42,A -85,B 0,C 180,E1 20105.377,E2 20105.377} C_VEL
LIN {X 0,Y 459.595,Z 697.97,A -85,B 0,C 180,E1 20101.621,E2 20101.621} C_VEL
LIN {X 0,Y 458.991,Z 708.731,A -85,B 0,C 180,E1 20100.685,E2 20100.685} C_VEL
LIN {X 0,Y 462.194,Z 733.446,A -85,B 0,C 180,E1 20100.056,E2 20100.056} C_VEL
LIN {X 0,Y 459.422,Z 922.267,A -85,B 0,C 180,E1 20097.007,E2 20097.007} C_VEL
LIN {X 0,Y 458.611,Z 941.638,A -85,B 0,C 180,E1 20096.473,E2 20096.473} C_VEL
LIN {X 0,Y 457.577,Z 960.021,A -85,B 0,C 180,E1 20095.74,E2 20095.74} C_VEL
LIN {X 0,Y 456.393,Z 977.811,A -85,B 0,C 180,E1 20094.8,E2 20094.8} C_VEL
LIN {X 0,Y 455.084,Z 995.368,A -85,B 0,C 180,E1 20093.626,E2 20093.626} C_VEL
LIN {X 0,Y 453.732,Z 1012.038,A -85,B 0,C 180,E1 20092.252,E2 20092.252} C_VEL
LIN {X 0,Y 452.446,Z 1027.533,A -85,B 0,C 180,E1 20090.706,E2 20090.706} C_VEL
LIN {X 0,Y 451.242,Z 1042.253,A -85,B 0,C 180,E1 20088.942,E2 20088.942} C_VEL
LIN {X 0,Y 450.217,Z 1055.46,A -85,B 0,C 180,E1 20087.046,E2 20087.046} C_VEL
LIN {X 0,Y 449.435,Z 1066.883,A -85,B 0,C 180,E1 20085.087,E2 20085.087} C_VEL
LIN {X 0,Y 448.829,Z 1076.979,A -85,B 0,C 180,E1 20083.002,E2 20083.002} C_VEL
LIN {X 0,Y 448.439,Z 1085.684,A -85,B 0,C 180,E1 20080.794,E2 20080.794} C_VEL
LIN {X 0,Y 448.193,Z 1092.889,A -85,B 0,C 180,E1 20078.467,E2 20078.467} C_VEL
LIN {X 0,Y 448.088,Z 1098.229,A -85,B 0,C 180,E1 20076.148,E2 20076.148} C_VEL
LIN {X 0,Y 448.068,Z 1101.96,A -85,B 0,C 180,E1 20073.71,E2 20073.71} C_VEL
LIN {X 0,Y 448.075,Z 1103.834,A -85,B 0,C 180,E1 20071.278,E2 20071.278} C_VEL
LIN {X 0,Y 448.076,Z 1103.908,A -85,B 0,C 180,E1 20068.977,E2 20068.977} C_VEL
LIN {X 0,Y 448.07,Z 1102.361,A -85,B 0,C 180,E1 20066.674,E2 20066.674} C_VEL
LIN {X 0,Y 448.079,Z 1099.165,A -85,B 0,C 180,E1 20064.365,E2 20064.365} C_VEL
LIN {X 0,Y 448.155,Z 1094.248,A -85,B 0,C 180,E1 20062.049,E2 20062.049} C_VEL
LIN {X 0,Y 448.363,Z 1087.504,A -85,B 0,C 180,E1 20059.723,E2 20059.723} C_VEL
LIN {X 0,Y 448.743,Z 1078.756,A -85,B 0,C 180,E1 20057.387,E2 20057.387} C_VEL
LIN {X 0,Y 449.348,Z 1068.412,A -85,B 0,C 180,E1 20055.173,E2 20055.173} C_VEL
LIN {X 0,Y 450.164,Z 1056.514,A -85,B 0,C 180,E1 20053.084,E2 20053.084} C_VEL
LIN {X 0,Y 451.174,Z 1043.539,A -85,B 0,C 180,E1 20051.189,E2 20051.189} C_VEL
LIN {X 0,Y 452.37,Z 1029.087,A -85,B 0,C 180,E1 20049.425,E2 20049.425} C_VEL
LIN {X 0,Y 453.663,Z 1013.701,A -85,B 0,C 180,E1 20047.859,E2 20047.859} C_VEL
LIN {X 0,Y 454.983,Z 997.654,A -85,B 0,C 180,E1 20046.507,E2 20046.507} C_VEL
LIN {X 0,Y 456.285,Z 980.52,A -85,B 0,C 180,E1 20045.326,E2 20045.326} C_VEL
LIN {X 0,Y 457.5,Z 962.835,A -85,B 0,C 180,E1 20044.359,E2 20044.359} C_VEL
LIN {X 0,Y 458.578,Z 943.936,A -85,B 0,C 180,E1 20043.577,E2 20043.577} C_VEL
LIN {X 0,Y 459.412,Z 924.752,A -85,B 0,C 180,E1 20043.024,E2 20043.024} C_VEL
LIN {X 0,Y 459.972,Z 893.91,A -85,B 0,C 180,E1 20042.492,E2 20042.492} C_VEL
LIN {X 0,Y 462.064,Z 730.77,A -85,B 0,C 180,E1 20039.882,E2 20039.882} C_VEL
LIN {X 0,Y 458.946,Z 708.201,A -85,B 0,C 180,E1 20039.292,E2 20039.292} C_VEL
LIN {X 0,Y 461.768,Z 667.955,A -85,B 0,C 180,E1 20035.663,E2 20035.663} C_VEL
LIN {X 0,Y 462.522,Z 656.289,A -85,B 0,C 180,E1 20034.585,E2 20034.585} C_VEL
LIN {X 0,Y 454.891,Z 634.362,A -85,B 0,C 180,E1 20031.794,E2 20031.794} C_VEL
LIN {X 0,Y 449.15,Z 618.534,A -85,B 0,C 180,E1 20029.581,E2 20029.581} C_VEL
LIN {X 0,Y 449.134,Z 618.284,A -85,B 0,C 180,E1 20026.006,E2 20026.006} C_VEL
LIN {X 0,Y 449.129,Z 618.288,A -85,B 0,C 180,E1 20022.246,E2 20022.246} C_VEL
LIN {X 0,Y 449.129,Z 618.286,A -85,B 0,C 180,E1 20018.56,E2 20018.56} C_VEL
LIN {X 0,Y 449.133,Z 618.29,A -85,B 0,C 180,E1 20014.767,E2 20014.767} C_VEL
LIN {X 0,Y 449.133,Z 618.289,A -85,B 0,C 180,E1 20010.947,E2 20010.947} C_VEL
LIN {X 0,Y 449.13,Z 618.287,A -85,B 0,C 180,E1 20007.297,E2 20007.297} C_VEL
LIN {X 0,Y 449.109,Z 618.291,A -85,B 0,C 180,E1 20003.624,E2 20003.624} C_VEL
LIN {X 0,Y 449.111,Z 618.295,A -85,B 0,C 180,E1 19999.915,E2 19999.915} C_VEL
LIN {X 0,Y 449.136,Z 618.292,A -85,B 0,C 180,E1 19996.29,E2 19996.29} C_VEL
LIN {X 0,Y 449.128,Z 618.292,A -85,B 0,C 180,E1 19992.601,E2 19992.601} C_VEL
LIN {X 0,Y 449.168,Z 618.526,A -85,B 0,C 180,E1 19990.354,E2 19990.354} C_VEL
LIN {X 0,Y 454.123,Z 634.459,A -85,B 0,C 180,E1 19988.164,E2 19988.164} C_VEL
LIN {X 0,Y 456.573,Z 644.548,A -85,B 0,C 180,E1 19986.854,E2 19986.854} C_VEL
LIN {X 0,Y 456.307,Z 677.879,A -85,B 0,C 180,E1 19983.077,E2 19983.077} C_VEL
LIN {X 0,Y 455.852,Z 706.351,A -85,B 0,C 180,E1 19979.748,E2 19979.748} C_VEL
LIN {X 0,Y 455.877,Z 711.904,A -85,B 0,C 180,E1 19979.148,E2 19979.148} C_VEL
LIN {X 0,Y 456.234,Z 715.899,A -85,B 0,C 180,E1 19979.048,E2 19979.048} C_VEL
LIN {X 0,Y 454.26,Z 849.577,A -85,B 0,C 180,E1 19976.656,E2 19976.656} C_VEL
LIN {X 0,Y 454.119,Z 865.595,A -85,B 0,C 180,E1 19976.157,E2 19976.157} C_VEL
LIN {X 0,Y 453.727,Z 881.903,A -85,B 0,C 180,E1 19975.386,E2 19975.386} C_VEL
LIN {X 0,Y 453.237,Z 895.864,A -85,B 0,C 180,E1 19974.493,E2 19974.493} C_VEL
LIN {X 0,Y 452.59,Z 909.755,A -85,B 0,C 180,E1 19973.339,E2 19973.339} C_VEL
LIN {X 0,Y 451.915,Z 922.058,A -85,B 0,C 180,E1 19972.051,E2 19972.051} C_VEL
LIN {X 0,Y 451.164,Z 933.986,A -85,B 0,C 180,E1 19970.472,E2 19970.472} C_VEL
LIN {X 0,Y 450.526,Z 943.631,A -85,B 0,C 180,E1 19968.867,E2 19968.867} C_VEL
LIN {X 0,Y 449.955,Z 952.269,A -85,B 0,C 180,E1 19967.03,E2 19967.03} C_VEL
LIN {X 0,Y 449.537,Z 958.919,A -85,B 0,C 180,E1 19965.18,E2 19965.18} C_VEL
LIN {X 0,Y 449.194,Z 964.397,A -85,B 0,C 180,E1 19963.046,E2 19963.046} C_VEL
LIN {X 0,Y 448.993,Z 967.647,A -85,B 0,C 180,E1 19961.026,E2 19961.026} C_VEL
LIN {X 0,Y 448.888,Z 969.236,A -85,B 0,C 180,E1 19958.848,E2 19958.848} C_VEL
LIN {X 0,Y 448.864,Z 968.89,A -85,B 0,C 180,E1 19956.779,E2 19956.779} C_VEL
LIN {X 0,Y 448.916,Z 966.78,A -85,B 0,C 180,E1 19954.682,E2 19954.682} C_VEL
LIN {X 0,Y 449.056,Z 962.972,A -85,B 0,C 180,E1 19952.675,E2 19952.675} C_VEL
LIN {X 0,Y 449.318,Z 957.402,A -85,B 0,C 180,E1 19950.688,E2 19950.688} C_VEL
LIN {X 0,Y 449.688,Z 950.162,A -85,B 0,C 180,E1 19948.797,E2 19948.797} C_VEL
LIN {X 0,Y 450.214,Z 941.053,A -85,B 0,C 180,E1 19946.958,E2 19946.958} C_VEL
LIN {X 0,Y 450.798,Z 931.087,A -85,B 0,C 180,E1 19945.374,E2 19945.374} C_VEL
LIN {X 0,Y 451.509,Z 918.943,A -85,B 0,C 180,E1 19943.821,E2 19943.821} C_VEL
LIN {X 0,Y 452.191,Z 905.782,A -85,B 0,C 180,E1 19942.492,E2 19942.492} C_VEL
LIN {X 0,Y 452.82,Z 892.405,A -85,B 0,C 180,E1 19941.413,E2 19941.413} C_VEL
LIN {X 0,Y 453.365,Z 877.507,A -85,B 0,C 180,E1 19940.486,E2 19940.486} C_VEL
LIN {X 0,Y 453.799,Z 861.05,A -85,B 0,C 180,E1 19939.734,E2 19939.734} C_VEL
LIN {X 0,Y 453.997,Z 844.32,A -85,B 0,C 180,E1 19939.24,E2 19939.24} C_VEL
LIN {X 0,Y 455.191,Z 746.791,A -85,B 0,C 180,E1 19937.57,E2 19937.57} C_VEL
LIN {X 0,Y 454.439,Z 738.103,A -85,B 0,C 180,E1 19937.38,E2 19937.38} C_VEL
LIN {X 0,Y 450.32,Z 722.316,A -85,B 0,C 180,E1 19936.904,E2 19936.904} C_VEL
LIN {X 0,Y 447.937,Z 712.776,A -85,B 0,C 180,E1 19936.617,E2 19936.617} C_VEL
LIN {X 0,Y 446.742,Z 706.166,A -85,B 0,C 180,E1 19936.41,E2 19936.41} C_VEL
LIN {X 0,Y 447.505,Z 675.537,A -85,B 0,C 180,E1 19932.685,E2 19932.685} C_VEL
LIN {X 0,Y 448.201,Z 646.371,A -85,B 0,C 180,E1 19929.148,E2 19929.148} C_VEL
LIN {X 0,Y 444.704,Z 631.781,A -85,B 0,C 180,E1 19927.135,E2 19927.135} C_VEL
LIN {X 0,Y 441.188,Z 619.451,A -85,B 0,C 180,E1 19925.345,E2 19925.345} C_VEL
LIN {X 0,Y 441.183,Z 619.281,A -85,B 0,C 180,E1 19921.722,E2 19921.722} C_VEL
LIN {X 0,Y 441.145,Z 619.281,A -85,B 0,C 180,E1 19918.128,E2 19918.128} C_VEL
LIN {X 0,Y 441.139,Z 619.251,A -85,B 0,C 180,E1 19914.335,E2 19914.335} C_VEL
LIN {X 0,Y 441.17,Z 619.262,A -85,B 0,C 180,E1 19910.705,E2 19910.705} C_VEL
LIN {X 0,Y 441.207,Z 619.523,A -85,B 0,C 180,E1 19907.39,E2 19907.39} C_VEL
LIN {X 0,Y 446.186,Z 636.822,A -85,B 0,C 180,E1 19904.271,E2 19904.271} C_VEL
LIN {X 0,Y 449.603,Z 650.544,A -85,B 0,C 180,E1 19901.936,E2 19901.936} C_VEL
LIN {X 0,Y 447.682,Z 677.48,A -85,B 0,C 180,E1 19898.089,E2 19898.089} C_VEL
LIN {X 0,Y 446.636,Z 694.549,A -85,B 0,C 180,E1 19895.718,E2 19895.718} C_VEL
LIN {X 0,Y 451,Z 716.632,A -85,B 0,C 180,E1 19895.062,E2 19895.062} C_VEL
LIN {X 0,Y 449.168,Z 842.476,A -85,B 0,C 180,E1 19892.96,E2 19892.96} C_VEL
LIN {X 0,Y 448.727,Z 859.47,A -85,B 0,C 180,E1 19892.427,E2 19892.427} C_VEL
LIN {X 0,Y 448.084,Z 875.224,A -85,B 0,C 180,E1 19891.698,E2 19891.698} C_VEL
LIN {X 0,Y 447.24,Z 889.986,A -85,B 0,C 180,E1 19890.769,E2 19890.769} C_VEL
LIN {X 0,Y 446.209,Z 904.96,A -85,B 0,C 180,E1 19889.551,E2 19889.551} C_VEL
LIN {X 0,Y 445.197,Z 918.043,A -85,B 0,C 180,E1 19888.199,E2 19888.199} C_VEL
LIN {X 0,Y 444.173,Z 930.061,A -85,B 0,C 180,E1 19886.645,E2 19886.645} C_VEL
LIN {X 0,Y 443.241,Z 940.614,A -85,B 0,C 180,E1 19884.953,E2 19884.953} C_VEL
LIN {X 0,Y 442.442,Z 949.635,A -85,B 0,C 180,E1 19883.121,E2 19883.121} C_VEL
LIN {X 0,Y 441.818,Z 957.22,A -85,B 0,C 180,E1 19881.148,E2 19881.148} C_VEL
LIN {X 0,Y 441.399,Z 962.948,A -85,B 0,C 180,E1 19879.164,E2 19879.164} C_VEL
LIN {X 0,Y 441.114,Z 967.185,A -85,B 0,C 180,E1 19877.033,E2 19877.033} C_VEL
LIN {X 0,Y 440.979,Z 969.711,A -85,B 0,C 180,E1 19874.886,E2 19874.886} C_VEL
LIN {X 0,Y 440.956,Z 970.511,A -85,B 0,C 180,E1 19872.672,E2 19872.672} C_VEL
LIN {X 0,Y 441.055,Z 969.492,A -85,B 0,C 180,E1 19870.397,E2 19870.397} C_VEL
LIN {X 0,Y 441.291,Z 966.836,A -85,B 0,C 180,E1 19868.275,E2 19868.275} C_VEL
LIN {X 0,Y 441.68,Z 962.219,A -85,B 0,C 180,E1 19866.096,E2 19866.096} C_VEL
LIN {X 0,Y 442.277,Z 955.859,A -85,B 0,C 180,E1 19863.987,E2 19863.987} C_VEL
LIN {X 0,Y 443.071,Z 947.786,A -85,B 0,C 180,E1 19862.006,E2 19862.006} C_VEL
LIN {X 0,Y 444.066,Z 938.177,A -85,B 0,C 180,E1 19860.159,E2 19860.159} C_VEL
LIN {X 0,Y 445.165,Z 927.224,A -85,B 0,C 180,E1 19858.492,E2 19858.492} C_VEL
LIN {X 0,Y 446.297,Z 915.157,A -85,B 0,C 180,E1 19857.016,E2 19857.016} C_VEL
LIN {X 0,Y 447.43,Z 902.065,A -85,B 0,C 180,E1 19855.727,E2 19855.727} C_VEL
LIN {X 0,Y 448.437,Z 888.204,A -85,B 0,C 180,E1 19854.649,E2 19854.649} C_VEL
LIN {X 0,Y 449.374,Z 872.554,A -85,B 0,C 180,E1 19853.712,E2 19853.712} C_VEL
LIN {X 0,Y 450.057,Z 856.42,A -85,B 0,C 180,E1 19853.008,E2 19853.008} C_VEL
LIN {X 0,Y 450.437,Z 839.487,A -85,B 0,C 180,E1 19852.535,E2 19852.535} C_VEL
LIN {X 0,Y 452.383,Z 715.551,A -85,B 0,C 180,E1 19850.415,E2 19850.415} C_VEL
LIN {X 0,Y 447.834,Z 695.278,A -85,B 0,C 180,E1 19849.708,E2 19849.708} C_VEL
LIN {X 0,Y 447.985,Z 691.048,A -85,B 0,C 180,E1 19849.16,E2 19849.16} C_VEL
LIN {X 0,Y 450.17,Z 664.54,A -85,B 0,C 180,E1 19845.296,E2 19845.296} C_VEL
LIN {X 0,Y 451.167,Z 652.821,A -85,B 0,C 180,E1 19843.558,E2 19843.558} C_VEL
LIN {X 0,Y 447.144,Z 637.825,A -85,B 0,C 180,E1 19840.764,E2 19840.764} C_VEL
LIN {X 0,Y 442.819,Z 624.413,A -85,B 0,C 180,E1 19838.055,E2 19838.055} C_VEL
LIN {X 0,Y 441.205,Z 619.397,A -85,B 0,C 180,E1 19836.955,E2 19836.955} C_VEL
LIN {X 0,Y 441.189,Z 619.277,A -85,B 0,C 180,E1 19833.105,E2 19833.105} C_VEL
LIN {X 0,Y 441.2,Z 619.274,A -85,B 0,C 180,E1 19829.308,E2 19829.308} C_VEL
LIN {X 0,Y 441.187,Z 619.269,A -85,B 0,C 180,E1 19825.506,E2 19825.506} C_VEL
LIN {X 0,Y 441.187,Z 619.271,A -85,B 0,C 180,E1 19821.679,E2 19821.679} C_VEL
LIN {X 0,Y 441.193,Z 619.269,A -85,B 0,C 180,E1 19817.857,E2 19817.857} C_VEL
LIN {X 0,Y 441.19,Z 619.265,A -85,B 0,C 180,E1 19814.034,E2 19814.034} C_VEL
LIN {X 0,Y 441.191,Z 619.264,A -85,B 0,C 180,E1 19810.314,E2 19810.314} C_VEL
LIN {X 0,Y 441.188,Z 619.27,A -85,B 0,C 180,E1 19806.507,E2 19806.507} C_VEL
LIN {X 0,Y 441.18,Z 619.277,A -85,B 0,C 180,E1 19802.728,E2 19802.728} C_VEL
LIN {X 0,Y 441.192,Z 619.276,A -85,B 0,C 180,E1 19798.961,E2 19798.961} C_VEL
LIN {X 0,Y 441.191,Z 619.261,A -85,B 0,C 180,E1 19795.19,E2 19795.19} C_VEL
LIN {X 0,Y 441.195,Z 619.263,A -85,B 0,C 180,E1 19791.398,E2 19791.398} C_VEL
LIN {X 0,Y 441.189,Z 619.273,A -85,B 0,C 180,E1 19787.567,E2 19787.567} C_VEL
LIN {X 0,Y 441.177,Z 619.279,A -85,B 0,C 180,E1 19783.814,E2 19783.814} C_VEL
LIN {X 0,Y 441.181,Z 619.275,A -85,B 0,C 180,E1 19779.988,E2 19779.988} C_VEL
LIN {X 0,Y 441.194,Z 619.265,A -85,B 0,C 180,E1 19776.286,E2 19776.286} C_VEL
LIN {X 0,Y 441.196,Z 619.265,A -85,B 0,C 180,E1 19772.464,E2 19772.464} C_VEL
LIN {X 0,Y 441.191,Z 619.264,A -85,B 0,C 180,E1 19768.691,E2 19768.691} C_VEL
LIN {X 0,Y 441.171,Z 619.271,A -85,B 0,C 180,E1 19765.013,E2 19765.013} C_VEL
LIN {X 0,Y 441.178,Z 619.276,A -85,B 0,C 180,E1 19761.225,E2 19761.225} C_VEL
LIN {X 0,Y 441.196,Z 619.282,A -85,B 0,C 180,E1 19757.52,E2 19757.52} C_VEL
LIN {X 0,Y 441.197,Z 619.272,A -85,B 0,C 180,E1 19753.703,E2 19753.703} C_VEL
LIN {X 0,Y 441.237,Z 619.553,A -85,B 0,C 180,E1 19751.722,E2 19751.722} C_VEL
LIN {X 0,Y 447.67,Z 636.063,A -85,B 0,C 180,E1 19749.038,E2 19749.038} C_VEL
LIN {X 0,Y 453.87,Z 654.082,A -85,B 0,C 180,E1 19746.479,E2 19746.479} C_VEL
LIN {X 0,Y 455.67,Z 659.937,A -85,B 0,C 180,E1 19745.709,E2 19745.709} C_VEL
LIN {X 0,Y 452.184,Z 700.412,A -85,B 0,C 180,E1 19741.887,E2 19741.887} C_VEL
LIN {X 0,Y 451.691,Z 708.536,A -85,B 0,C 180,E1 19741.17,E2 19741.17} C_VEL
LIN {X 0,Y 455.011,Z 734.469,A -85,B 0,C 180,E1 19740.486,E2 19740.486} C_VEL
LIN {X 0,Y 452.07,Z 921.328,A -85,B 0,C 180,E1 19737.416,E2 19737.416} C_VEL
LIN {X 0,Y 451.197,Z 940.924,A -85,B 0,C 180,E1 19736.867,E2 19736.867} C_VEL
LIN {X 0,Y 450.109,Z 959.105,A -85,B 0,C 180,E1 19736.132,E2 19736.132} C_VEL
LIN {X 0,Y 448.801,Z 977.572,A -85,B 0,C 180,E1 19735.135,E2 19735.135} C_VEL
LIN {X 0,Y 447.403,Z 995.122,A -85,B 0,C 180,E1 19733.931,E2 19733.931} C_VEL
LIN {X 0,Y 445.97,Z 1011.719,A -85,B 0,C 180,E1 19732.528,E2 19732.528} C_VEL
LIN {X 0,Y 444.565,Z 1027.701,A -85,B 0,C 180,E1 19730.884,E2 19730.884} C_VEL
LIN {X 0,Y 443.316,Z 1042.218,A -85,B 0,C 180,E1 19729.089,E2 19729.089} C_VEL
LIN {X 0,Y 442.225,Z 1055.656,A -85,B 0,C 180,E1 19727.093,E2 19727.093} C_VEL
LIN {X 0,Y 441.389,Z 1067.531,A -85,B 0,C 180,E1 19724.965,E2 19724.965} C_VEL
LIN {X 0,Y 440.775,Z 1077.848,A -85,B 0,C 180,E1 19722.711,E2 19722.711} C_VEL
LIN {X 0,Y 440.425,Z 1086.133,A -85,B 0,C 180,E1 19720.464,E2 19720.464} C_VEL
LIN {X 0,Y 440.221,Z 1092.941,A -85,B 0,C 180,E1 19718.095,E2 19718.095} C_VEL
LIN {X 0,Y 440.155,Z 1097.904,A -85,B 0,C 180,E1 19715.736,E2 19715.736} C_VEL
LIN {X 0,Y 440.154,Z 1101.137,A -85,B 0,C 180,E1 19713.386,E2 19713.386} C_VEL
LIN {X 0,Y 440.165,Z 1102.712,A -85,B 0,C 180,E1 19711.041,E2 19711.041} C_VEL
LIN {X 0,Y 440.16,Z 1102.656,A -85,B 0,C 180,E1 19708.698,E2 19708.698} C_VEL
LIN {X 0,Y 440.143,Z 1100.927,A -85,B 0,C 180,E1 19706.353,E2 19706.353} C_VEL
LIN {X 0,Y 440.146,Z 1097.522,A -85,B 0,C 180,E1 19704.002,E2 19704.002} C_VEL
LIN {X 0,Y 440.223,Z 1092.383,A -85,B 0,C 180,E1 19701.641,E2 19701.641} C_VEL
LIN {X 0,Y 440.445,Z 1085.401,A -85,B 0,C 180,E1 19699.272,E2 19699.272} C_VEL
LIN {X 0,Y 440.825,Z 1076.936,A -85,B 0,C 180,E1 19697.023,E2 19697.023} C_VEL
LIN {X 0,Y 441.43,Z 1067.097,A -85,B 0,C 180,E1 19694.901,E2 19694.901} C_VEL
LIN {X 0,Y 442.295,Z 1055.152,A -85,B 0,C 180,E1 19692.774,E2 19692.774} C_VEL
LIN {X 0,Y 443.419,Z 1041.636,A -85,B 0,C 180,E1 19690.779,E2 19690.779} C_VEL
LIN {X 0,Y 444.698,Z 1027.019,A -85,B 0,C 180,E1 19688.984,E2 19688.984} C_VEL
LIN {X 0,Y 446.076,Z 1011.495,A -85,B 0,C 180,E1 19687.399,E2 19687.399} C_VEL
LIN {X 0,Y 447.516,Z 994.909,A -85,B 0,C 180,E1 19686.006,E2 19686.006} C_VEL
LIN {X 0,Y 448.903,Z 977.533,A -85,B 0,C 180,E1 19684.822,E2 19684.822} C_VEL
LIN {X 0,Y 450.196,Z 959.236,A -85,B 0,C 180,E1 19683.841,E2 19683.841} C_VEL
LIN {X 0,Y 451.338,Z 939.908,A -85,B 0,C 180,E1 19683.069,E2 19683.069} C_VEL
LIN {X 0,Y 452.179,Z 920.059,A -85,B 0,C 180,E1 19682.537,E2 19682.537} C_VEL
LIN {X 0,Y 454.827,Z 731.839,A -85,B 0,C 180,E1 19679.466,E2 19679.466} C_VEL
LIN {X 0,Y 451.572,Z 707.948,A -85,B 0,C 180,E1 19678.831,E2 19678.831} C_VEL
LIN {X 0,Y 454.671,Z 666.766,A -85,B 0,C 180,E1 19675.057,E2 19675.057} C_VEL
LIN {X 0,Y 455.267,Z 659.247,A -85,B 0,C 180,E1 19674.35,E2 19674.35} C_VEL
LIN {X 0,Y 447.7,Z 637.342,A -85,B 0,C 180,E1 19671.516,E2 19671.516} C_VEL
LIN {X 0,Y 441.229,Z 619.473,A -85,B 0,C 180,E1 19668.953,E2 19668.953} C_VEL
LIN {X 0,Y 441.188,Z 619.278,A -85,B 0,C 180,E1 19665.182,E2 19665.182} C_VEL
LIN {X 0,Y 441.186,Z 619.274,A -85,B 0,C 180,E1 19661.396,E2 19661.396} C_VEL
LIN {X 0,Y 441.196,Z 619.276,A -85,B 0,C 180,E1 19657.726,E2 19657.726} C_VEL
LIN {X 0,Y 441.184,Z 619.279,A -85,B 0,C 180,E1 19653.884,E2 19653.884} C_VEL
LIN {X 0,Y 441.177,Z 619.28,A -85,B 0,C 180,E1 19650.057,E2 19650.057} C_VEL
LIN {X 0,Y 441.19,Z 619.28,A -85,B 0,C 180,E1 19646.371,E2 19646.371} C_VEL
LIN {X 0,Y 441.203,Z 619.278,A -85,B 0,C 180,E1 19642.519,E2 19642.519} C_VEL
LIN {X 0,Y 441.2,Z 619.278,A -85,B 0,C 180,E1 19638.686,E2 19638.686} C_VEL
LIN {X 0,Y 441.169,Z 619.283,A -85,B 0,C 180,E1 19634.973,E2 19634.973} C_VEL
LIN {X 0,Y 441.155,Z 619.285,A -85,B 0,C 180,E1 19631.24,E2 19631.24} C_VEL
LIN {X 0,Y 441.208,Z 619.605,A -85,B 0,C 180,E1 19630.907,E2 19630.907} C_VEL
LIN {X 0,Y 446.641,Z 636.354,A -85,B 0,C 180,E1 19628.561,E2 19628.561} C_VEL
LIN {X 0,Y 449.304,Z 646.976,A -85,B 0,C 180,E1 19627.159,E2 19627.159} C_VEL
LIN {X 0,Y 449.067,Z 676.196,A -85,B 0,C 180,E1 19623.83,E2 19623.83} C_VEL
LIN {X 0,Y 448.583,Z 704.636,A -85,B 0,C 180,E1 19620.511,E2 19620.511} C_VEL
LIN {X 0,Y 448.528,Z 713.229,A -85,B 0,C 180,E1 19619.533,E2 19619.533} C_VEL
LIN {X 0,Y 448.876,Z 717.187,A -85,B 0,C 180,E1 19619.431,E2 19619.431} C_VEL
LIN {X 0,Y 446.74,Z 850.597,A -85,B 0,C 180,E1 19616.985,E2 19616.985} C_VEL
LIN {X 0,Y 446.599,Z 866.734,A -85,B 0,C 180,E1 19616.478,E2 19616.478} C_VEL
LIN {X 0,Y 446.194,Z 882.908,A -85,B 0,C 180,E1 19615.704,E2 19615.704} C_VEL
LIN {X 0,Y 445.67,Z 897.077,A -85,B 0,C 180,E1 19614.787,E2 19614.787} C_VEL
LIN {X 0,Y 444.98,Z 910.966,A -85,B 0,C 180,E1 19613.614,E2 19613.614} C_VEL
LIN {X 0,Y 444.26,Z 923.284,A -85,B 0,C 180,E1 19612.304,E2 19612.304} C_VEL
LIN {X 0,Y 443.497,Z 934.615,A -85,B 0,C 180,E1 19610.789,E2 19610.789} C_VEL
LIN {X 0,Y 442.82,Z 944.32,A -85,B 0,C 180,E1 19609.176,E2 19609.176} C_VEL
LIN {X 0,Y 442.194,Z 952.987,A -85,B 0,C 180,E1 19607.33,E2 19607.33} C_VEL
LIN {X 0,Y 441.732,Z 959.794,A -85,B 0,C 180,E1 19605.448,E2 19605.448} C_VEL
LIN {X 0,Y 441.355,Z 965.126,A -85,B 0,C 180,E1 19603.393,E2 19603.393} C_VEL
LIN {X 0,Y 441.129,Z 968.612,A -85,B 0,C 180,E1 19601.342,E2 19601.342} C_VEL
LIN {X 0,Y 440.994,Z 970.351,A -85,B 0,C 180,E1 19599.147,E2 19599.147} C_VEL
LIN {X 0,Y 440.955,Z 970.243,A -85,B 0,C 180,E1 19597.015,E2 19597.015} C_VEL
LIN {X 0,Y 441.001,Z 968.135,A -85,B 0,C 180,E1 19594.77,E2 19594.77} C_VEL
LIN {X 0,Y 441.148,Z 964.492,A -85,B 0,C 180,E1 19592.752,E2 19592.752} C_VEL
LIN {X 0,Y 441.42,Z 958.921,A -85,B 0,C 180,E1 19590.7,E2 19590.7} C_VEL
LIN {X 0,Y 441.81,Z 951.832,A -85,B 0,C 180,E1 19588.785,E2 19588.785} C_VEL
LIN {X 0,Y 442.38,Z 942.43,A -85,B 0,C 180,E1 19586.841,E2 19586.841} C_VEL
LIN {X 0,Y 443.016,Z 932.159,A -85,B 0,C 180,E1 19585.179,E2 19585.179} C_VEL
LIN {X 0,Y 443.736,Z 920.456,A -85,B 0,C 180,E1 19583.657,E2 19583.657} C_VEL
LIN {X 0,Y 444.421,Z 908.066,A -85,B 0,C 180,E1 19582.367,E2 19582.367} C_VEL
LIN {X 0,Y 445.119,Z 893.88,A -85,B 0,C 180,E1 19581.192,E2 19581.192} C_VEL
LIN {X 0,Y 445.686,Z 879.219,A -85,B 0,C 180,E1 19580.254,E2 19580.254} C_VEL
LIN {X 0,Y 446.146,Z 862.671,A -85,B 0,C 180,E1 19579.478,E2 19579.478} C_VEL
LIN {X 0,Y 446.356,Z 846.289,A -85,B 0,C 180,E1 19578.973,E2 19578.973} C_VEL
LIN {X 0,Y 448.001,Z 713.107,A -85,B 0,C 180,E1 19576.626,E2 19576.626} C_VEL
LIN {X 0,Y 447.937,Z 712.776,A -85,B 0,C 180,E1 19576.617,E2 19576.617} C_VEL
LIN {X 0,Y 446.632,Z 708.098,A -85,B 0,C 180,E1 19576.372,E2 19576.372} C_VEL
LIN {X 0,Y 444.247,Z 702.664,A -85,B 0,C 180,E1 19575.793,E2 19575.793} C_VEL
LIN {X 0,Y 440.608,Z 693.827,A -85,B 0,C 180,E1 19574.499,E2 19574.499} C_VEL
LIN {X 0,Y 439.767,Z 687.238,A -85,B 0,C 180,E1 19573.619,E2 19573.619} C_VEL
LIN {X 0,Y 440.488,Z 657.213,A -85,B 0,C 180,E1 19569.97,E2 19569.97} C_VEL
LIN {X 0,Y 440.567,Z 647.522,A -85,B 0,C 180,E1 19568.784,E2 19568.784} C_VEL
LIN {X 0,Y 435.793,Z 629.342,A -85,B 0,C 180,E1 19566.214,E2 19566.214} C_VEL
LIN {X 0,Y 433.223,Z 620.443,A -85,B 0,C 180,E1 19564.888,E2 19564.888} C_VEL
LIN {X 0,Y 433.24,Z 620.268,A -85,B 0,C 180,E1 19561.284,E2 19561.284} C_VEL
LIN {X 0,Y 433.244,Z 620.271,A -85,B 0,C 180,E1 19557.598,E2 19557.598} C_VEL
LIN {X 0,Y 433.215,Z 620.242,A -85,B 0,C 180,E1 19553.823,E2 19553.823} C_VEL
LIN {X 0,Y 433.206,Z 620.246,A -85,B 0,C 180,E1 19550.115,E2 19550.115} C_VEL
LIN {X 0,Y 433.25,Z 620.554,A -85,B 0,C 180,E1 19547.945,E2 19547.945} C_VEL
LIN {X 0,Y 438.334,Z 638.042,A -85,B 0,C 180,E1 19544.722,E2 19544.722} C_VEL
LIN {X 0,Y 442.147,Z 652.541,A -85,B 0,C 180,E1 19542.207,E2 19542.207} C_VEL
LIN {X 0,Y 440.065,Z 679.997,A -85,B 0,C 180,E1 19538.23,E2 19538.23} C_VEL
LIN {X 0,Y 439.13,Z 694.648,A -85,B 0,C 180,E1 19536.176,E2 19536.176} C_VEL
LIN {X 0,Y 443.709,Z 717.934,A -85,B 0,C 180,E1 19535.47,E2 19535.47} C_VEL
LIN {X 0,Y 441.777,Z 843.146,A -85,B 0,C 180,E1 19533.345,E2 19533.345} C_VEL
LIN {X 0,Y 441.312,Z 860.243,A -85,B 0,C 180,E1 19532.801,E2 19532.801} C_VEL
LIN {X 0,Y 440.653,Z 875.609,A -85,B 0,C 180,E1 19532.081,E2 19532.081} C_VEL
LIN {X 0,Y 439.739,Z 890.909,A -85,B 0,C 180,E1 19531.108,E2 19531.108} C_VEL
LIN {X 0,Y 438.651,Z 905.888,A -85,B 0,C 180,E1 19529.87,E2 19529.87} C_VEL
LIN {X 0,Y 437.63,Z 918.444,A -85,B 0,C 180,E1 19528.56,E2 19528.56} C_VEL
LIN {X 0,Y 436.536,Z 930.569,A -85,B 0,C 180,E1 19526.981,E2 19526.981} C_VEL
LIN {X 0,Y 435.536,Z 941.223,A -85,B 0,C 180,E1 19525.26,E2 19525.26} C_VEL
LIN {X 0,Y 434.677,Z 950.366,A -85,B 0,C 180,E1 19523.396,E2 19523.396} C_VEL
LIN {X 0,Y 433.967,Z 958.425,A -85,B 0,C 180,E1 19521.273,E2 19521.273} C_VEL
LIN {X 0,Y 433.513,Z 964.182,A -85,B 0,C 180,E1 19519.233,E2 19519.233} C_VEL
LIN {X 0,Y 433.21,Z 968.403,A -85,B 0,C 180,E1 19517.063,E2 19517.063} C_VEL
LIN {X 0,Y 433.066,Z 970.973,A -85,B 0,C 180,E1 19514.814,E2 19514.814} C_VEL
LIN {X 0,Y 433.046,Z 971.694,A -85,B 0,C 180,E1 19512.533,E2 19512.533} C_VEL
LIN {X 0,Y 433.161,Z 970.685,A -85,B 0,C 180,E1 19510.306,E2 19510.306} C_VEL
LIN {X 0,Y 433.415,Z 968.123,A -85,B 0,C 180,E1 19508.197,E2 19508.197} C_VEL
LIN {X 0,Y 433.819,Z 963.781,A -85,B 0,C 180,E1 19506.069,E2 19506.069} C_VEL
LIN {X 0,Y 434.452,Z 957.552,A -85,B 0,C 180,E1 19503.924,E2 19503.924} C_VEL
LIN {X 0,Y 435.236,Z 950.35,A -85,B 0,C 180,E1 19502.054,E2 19502.054} C_VEL
LIN {X 0,Y 436.256,Z 941.065,A -85,B 0,C 180,E1 19500.176,E2 19500.176} C_VEL
LIN {X 0,Y 437.438,Z 930.312,A -85,B 0,C 180,E1 19498.438,E2 19498.438} C_VEL
LIN {X 0,Y 438.635,Z 918.685,A -85,B 0,C 180,E1 19496.93,E2 19496.93} C_VEL
LIN {X 0,Y 439.889,Z 905.18,A -85,B 0,C 180,E1 19495.531,E2 19495.531} C_VEL
LIN {X 0,Y 441.039,Z 891.009,A -85,B 0,C 180,E1 19494.364,E2 19494.364} C_VEL
LIN {X 0,Y 442.02,Z 876.052,A -85,B 0,C 180,E1 19493.42,E2 19493.42} C_VEL
LIN {X 0,Y 442.813,Z 859.289,A -85,B 0,C 180,E1 19492.642,E2 19492.642} C_VEL
LIN {X 0,Y 443.269,Z 842.862,A -85,B 0,C 180,E1 19492.137,E2 19492.137} C_VEL
LIN {X 0,Y 445.396,Z 717.005,A -85,B 0,C 180,E1 19489.94,E2 19489.94} C_VEL
LIN {X 0,Y 440.523,Z 695.397,A -85,B 0,C 180,E1 19489.159,E2 19489.159} C_VEL
LIN {X 0,Y 440.867,Z 689.515,A -85,B 0,C 180,E1 19488.356,E2 19488.356} C_VEL
LIN {X 0,Y 443.152,Z 663.667,A -85,B 0,C 180,E1 19484.523,E2 19484.523} C_VEL
LIN {X 0,Y 443.773,Z 655.201,A -85,B 0,C 180,E1 19483.231,E2 19483.231} C_VEL
LIN {X 0,Y 439.757,Z 640.301,A -85,B 0,C 180,E1 19480.388,E2 19480.388} C_VEL
LIN {X 0,Y 435.304,Z 626.299,A -85,B 0,C 180,E1 19477.495,E2 19477.495} C_VEL
LIN {X 0,Y 433.262,Z 620.365,A -85,B 0,C 180,E1 19476.127,E2 19476.127} C_VEL
LIN {X 0,Y 433.254,Z 620.267,A -85,B 0,C 180,E1 19472.366,E2 19472.366} C_VEL
LIN {X 0,Y 433.254,Z 620.259,A -85,B 0,C 180,E1 19468.536,E2 19468.536} C_VEL
LIN {X 0,Y 433.25,Z 620.261,A -85,B 0,C 180,E1 19464.691,E2 19464.691} C_VEL
LIN {X 0,Y 433.258,Z 620.264,A -85,B 0,C 180,E1 19460.818,E2 19460.818} C_VEL
LIN {X 0,Y 433.25,Z 620.266,A -85,B 0,C 180,E1 19457.043,E2 19457.043} C_VEL
LIN {X 0,Y 433.244,Z 620.265,A -85,B 0,C 180,E1 19453.208,E2 19453.208} C_VEL
LIN {X 0,Y 433.253,Z 620.255,A -85,B 0,C 180,E1 19449.431,E2 19449.431} C_VEL
LIN {X 0,Y 433.251,Z 620.253,A -85,B 0,C 180,E1 19445.695,E2 19445.695} C_VEL
LIN {X 0,Y 433.254,Z 620.262,A -85,B 0,C 180,E1 19441.852,E2 19441.852} C_VEL
LIN {X 0,Y 433.247,Z 620.265,A -85,B 0,C 180,E1 19438.149,E2 19438.149} C_VEL
LIN {X 0,Y 433.24,Z 620.264,A -85,B 0,C 180,E1 19434.305,E2 19434.305} C_VEL
LIN {X 0,Y 433.245,Z 620.251,A -85,B 0,C 180,E1 19430.569,E2 19430.569} C_VEL
LIN {X 0,Y 433.255,Z 620.254,A -85,B 0,C 180,E1 19426.793,E2 19426.793} C_VEL
LIN {X 0,Y 433.257,Z 620.267,A -85,B 0,C 180,E1 19422.957,E2 19422.957} C_VEL
LIN {X 0,Y 433.254,Z 620.265,A -85,B 0,C 180,E1 19419.172,E2 19419.172} C_VEL
LIN {X 0,Y 433.238,Z 620.268,A -85,B 0,C 180,E1 19415.409,E2 19415.409} C_VEL
LIN {X 0,Y 433.239,Z 620.264,A -85,B 0,C 180,E1 19411.557,E2 19411.557} C_VEL
LIN {X 0,Y 433.253,Z 620.26,A -85,B 0,C 180,E1 19407.785,E2 19407.785} C_VEL
LIN {X 0,Y 433.257,Z 620.264,A -85,B 0,C 180,E1 19403.951,E2 19403.951} C_VEL
LIN {X 0,Y 433.263,Z 620.268,A -85,B 0,C 180,E1 19400.093,E2 19400.093} C_VEL
LIN {X 0,Y 433.245,Z 620.26,A -85,B 0,C 180,E1 19396.249,E2 19396.249} C_VEL
LIN {X 0,Y 433.258,Z 620.471,A -85,B 0,C 180,E1 19392.58,E2 19392.58} C_VEL
LIN {X 0,Y 437.244,Z 630.47,A -85,B 0,C 180,E1 19390.808,E2 19390.808} C_VEL
LIN {X 0,Y 443.275,Z 646.55,A -85,B 0,C 180,E1 19388.284,E2 19388.284} C_VEL
LIN {X 0,Y 448.499,Z 662.692,A -85,B 0,C 180,E1 19386.03,E2 19386.03} C_VEL
LIN {X 0,Y 444.807,Z 702.558,A -85,B 0,C 180,E1 19382.19,E2 19382.19} C_VEL
LIN {X 0,Y 444.462,Z 708.457,A -85,B 0,C 180,E1 19381.674,E2 19381.674} C_VEL
LIN {X 0,Y 447.891,Z 735.604,A -85,B 0,C 180,E1 19380.937,E2 19380.937} C_VEL
LIN {X 0,Y 444.764,Z 920.658,A -85,B 0,C 180,E1 19377.842,E2 19377.842} C_VEL
LIN {X 0,Y 443.846,Z 940.003,A -85,B 0,C 180,E1 19377.292,E2 19377.292} C_VEL
LIN {X 0,Y 442.667,Z 958.475,A -85,B 0,C 180,E1 19376.529,E2 19376.529} C_VEL
LIN {X 0,Y 441.344,Z 976.054,A -85,B 0,C 180,E1 19375.567,E2 19375.567} C_VEL
LIN {X 0,Y 439.866,Z 993.398,A -85,B 0,C 180,E1 19374.366,E2 19374.366} C_VEL
LIN {X 0,Y 438.361,Z 1009.945,A -85,B 0,C 180,E1 19372.956,E2 19372.956} C_VEL
LIN {X 0,Y 436.913,Z 1025.59,A -85,B 0,C 180,E1 19371.337,E2 19371.337} C_VEL
LIN {X 0,Y 435.578,Z 1040.257,A -85,B 0,C 180,E1 19369.511,E2 19369.511} C_VEL
LIN {X 0,Y 434.437,Z 1053.415,A -85,B 0,C 180,E1 19367.547,E2 19367.547} C_VEL
LIN {X 0,Y 433.526,Z 1065.483,A -85,B 0,C 180,E1 19365.38,E2 19365.38} C_VEL
LIN {X 0,Y 432.89,Z 1075.423,A -85,B 0,C 180,E1 19363.218,E2 19363.218} C_VEL
LIN {X 0,Y 432.503,Z 1083.981,A -85,B 0,C 180,E1 19360.927,E2 19360.927} C_VEL
LIN {X 0,Y 432.292,Z 1090.714,A -85,B 0,C 180,E1 19358.646,E2 19358.646} C_VEL
LIN {X 0,Y 432.214,Z 1096.011,A -85,B 0,C 180,E1 19356.242,E2 19356.242} C_VEL
LIN {X 0,Y 432.223,Z 1099.551,A -85,B 0,C 180,E1 19353.846,E2 19353.846} C_VEL
LIN {X 0,Y 432.25,Z 1101.38,A -85,B 0,C 180,E1 19351.458,E2 19351.458} C_VEL
LIN {X 0,Y 432.253,Z 1101.562,A -85,B 0,C 180,E1 19349.072,E2 19349.072} C_VEL
LIN {X 0,Y 432.229,Z 1100.106,A -85,B 0,C 180,E1 19346.684,E2 19346.684} C_VEL
LIN {X 0,Y 432.209,Z 1096.986,A -85,B 0,C 180,E1 19344.291,E2 19344.291} C_VEL
LIN {X 0,Y 432.256,Z 1092.134,A -85,B 0,C 180,E1 19341.888,E2 19341.888} C_VEL
LIN {X 0,Y 432.443,Z 1085.446,A -85,B 0,C 180,E1 19339.475,E2 19339.475} C_VEL
LIN {X 0,Y 432.825,Z 1076.747,A -85,B 0,C 180,E1 19337.051,E2 19337.051} C_VEL
LIN {X 0,Y 433.474,Z 1066.45,A -85,B 0,C 180,E1 19334.754,E2 19334.754} C_VEL
LIN {X 0,Y 434.373,Z 1054.598,A -85,B 0,C 180,E1 19332.588,E2 19332.588} C_VEL
LIN {X 0,Y 435.463,Z 1042.066,A -85,B 0,C 180,E1 19330.681,E2 19330.681} C_VEL
LIN {X 0,Y 436.826,Z 1027.232,A -85,B 0,C 180,E1 19328.798,E2 19328.798} C_VEL
LIN {X 0,Y 438.273,Z 1011.772,A -85,B 0,C 180,E1 19327.171,E2 19327.171} C_VEL
LIN {X 0,Y 439.798,Z 995.203,A -85,B 0,C 180,E1 19325.735,E2 19325.735} C_VEL
LIN {X 0,Y 441.291,Z 977.63,A -85,B 0,C 180,E1 19324.501,E2 19324.501} C_VEL
LIN {X 0,Y 442.646,Z 959.612,A -85,B 0,C 180,E1 19323.505,E2 19323.505} C_VEL
LIN {X 0,Y 443.819,Z 941.032,A -85,B 0,C 180,E1 19322.735,E2 19322.735} C_VEL
LIN {X 0,Y 444.717,Z 921.881,A -85,B 0,C 180,E1 19322.186,E2 19322.186} C_VEL
LIN {X 0,Y 445.5,Z 874.101,A -85,B 0,C 180,E1 19321.375,E2 19321.375} C_VEL
LIN {X 0,Y 447.571,Z 732.816,A -85,B 0,C 180,E1 19319.044,E2 19319.044} C_VEL
LIN {X 0,Y 444.21,Z 707.824,A -85,B 0,C 180,E1 19318.368,E2 19318.368} C_VEL
LIN {X 0,Y 447.315,Z 669.405,A -85,B 0,C 180,E1 19314.781,E2 19314.781} C_VEL
LIN {X 0,Y 447.852,Z 661.678,A -85,B 0,C 180,E1 19314.043,E2 19314.043} C_VEL
LIN {X 0,Y 440.407,Z 640.141,A -85,B 0,C 180,E1 19311.199,E2 19311.199} C_VEL
LIN {X 0,Y 433.285,Z 620.473,A -85,B 0,C 180,E1 19308.323,E2 19308.323} C_VEL
LIN {X 0,Y 433.251,Z 620.266,A -85,B 0,C 180,E1 19304.553,E2 19304.553} C_VEL
LIN {X 0,Y 433.262,Z 620.265,A -85,B 0,C 180,E1 19300.775,E2 19300.775} C_VEL
LIN {X 0,Y 433.254,Z 620.27,A -85,B 0,C 180,E1 19297.013,E2 19297.013} C_VEL
LIN {X 0,Y 433.256,Z 620.268,A -85,B 0,C 180,E1 19293.157,E2 19293.157} C_VEL
LIN {X 0,Y 433.262,Z 620.264,A -85,B 0,C 180,E1 19289.269,E2 19289.269} C_VEL
LIN {X 0,Y 433.244,Z 620.268,A -85,B 0,C 180,E1 19285.42,E2 19285.42} C_VEL
LIN {X 0,Y 433.229,Z 620.27,A -85,B 0,C 180,E1 19281.67,E2 19281.67} C_VEL
LIN {X 0,Y 433.232,Z 620.271,A -85,B 0,C 180,E1 19277.875,E2 19277.875} C_VEL
LIN {X 0,Y 433.257,Z 620.27,A -85,B 0,C 180,E1 19274.159,E2 19274.159} C_VEL
LIN {X 0,Y 433.245,Z 620.458,A -85,B 0,C 180,E1 19271.582,E2 19271.582} C_VEL
LIN {X 0,Y 437.993,Z 634.322,A -85,B 0,C 180,E1 19269.535,E2 19269.535} C_VEL
LIN {X 0,Y 442.108,Z 649.783,A -85,B 0,C 180,E1 19267.439,E2 19267.439} C_VEL
LIN {X 0,Y 441.753,Z 682.41,A -85,B 0,C 180,E1 19263.698,E2 19263.698} C_VEL
LIN {X 0,Y 441.217,Z 711.596,A -85,B 0,C 180,E1 19260.259,E2 19260.259} C_VEL
LIN {X 0,Y 441.291,Z 714.84,A -85,B 0,C 180,E1 19259.931,E2 19259.931} C_VEL
LIN {X 0,Y 441.554,Z 718.983,A -85,B 0,C 180,E1 19259.825,E2 19259.825} C_VEL
LIN {X 0,Y 439.245,Z 851.242,A -85,B 0,C 180,E1 19257.337,E2 19257.337} C_VEL
LIN {X 0,Y 439.097,Z 867.893,A -85,B 0,C 180,E1 19256.81,E2 19256.81} C_VEL
LIN {X 0,Y 438.7,Z 883.1,A -85,B 0,C 180,E1 19256.079,E2 19256.079} C_VEL
LIN {X 0,Y 438.159,Z 897.423,A -85,B 0,C 180,E1 19255.156,E2 19255.156} C_VEL
LIN {X 0,Y 437.464,Z 910.84,A -85,B 0,C 180,E1 19254.031,E2 19254.031} C_VEL
LIN {X 0,Y 436.663,Z 924.019,A -85,B 0,C 180,E1 19252.633,E2 19252.633} C_VEL
LIN {X 0,Y 435.876,Z 935.016,A -85,B 0,C 180,E1 19251.159,E2 19251.159} C_VEL
LIN {X 0,Y 435.09,Z 945.482,A -85,B 0,C 180,E1 19249.406,E2 19249.406} C_VEL
LIN {X 0,Y 434.447,Z 953.709,A -85,B 0,C 180,E1 19247.641,E2 19247.641} C_VEL
LIN {X 0,Y 433.929,Z 960.63,A -85,B 0,C 180,E1 19245.726,E2 19245.726} C_VEL
LIN {X 0,Y 433.542,Z 965.767,A -85,B 0,C 180,E1 19243.796,E2 19243.796} C_VEL
LIN {X 0,Y 433.255,Z 969.653,A -85,B 0,C 180,E1 19241.568,E2 19241.568} C_VEL
LIN {X 0,Y 433.103,Z 971.479,A -85,B 0,C 180,E1 19239.457,E2 19239.457} C_VEL
LIN {X 0,Y 433.047,Z 971.571,A -85,B 0,C 180,E1 19237.32,E2 19237.32} C_VEL
LIN {X 0,Y 433.078,Z 969.863,A -85,B 0,C 180,E1 19235.153,E2 19235.153} C_VEL
LIN {X 0,Y 433.223,Z 966.253,A -85,B 0,C 180,E1 19232.956,E2 19232.956} C_VEL
LIN {X 0,Y 433.492,Z 960.93,A -85,B 0,C 180,E1 19230.877,E2 19230.877} C_VEL
LIN {X 0,Y 433.891,Z 954.08,A -85,B 0,C 180,E1 19228.923,E2 19228.923} C_VEL
LIN {X 0,Y 434.409,Z 945.752,A -85,B 0,C 180,E1 19227.099,E2 19227.099} C_VEL
LIN {X 0,Y 435.115,Z 935.086,A -85,B 0,C 180,E1 19225.257,E2 19225.257} C_VEL
LIN {X 0,Y 435.886,Z 923.051,A -85,B 0,C 180,E1 19223.625,E2 19223.625} C_VEL
LIN {X 0,Y 436.659,Z 910.073,A -85,B 0,C 180,E1 19222.218,E2 19222.218} C_VEL
LIN {X 0,Y 437.408,Z 895.462,A -85,B 0,C 180,E1 19220.976,E2 19220.976} C_VEL
LIN {X 0,Y 438.004,Z 880.983,A -85,B 0,C 180,E1 19220.022,E2 19220.022} C_VEL
LIN {X 0,Y 438.496,Z 864.122,A -85,B 0,C 180,E1 19219.21,E2 19219.21} C_VEL
LIN {X 0,Y 438.724,Z 847.92,A -85,B 0,C 180,E1 19218.694,E2 19218.694} C_VEL
LIN {X 0,Y 440.514,Z 714.271,A -85,B 0,C 180,E1 19216.279,E2 19216.279} C_VEL
LIN {X 0,Y 439.214,Z 707.032,A -85,B 0,C 180,E1 19216.045,E2 19216.045} C_VEL
LIN {X 0,Y 439.767,Z 687.238,A -85,B 0,C 180,E1 19213.619,E2 19213.619} C_VEL
LIN {X 0,Y 438.967,Z 681.843,A -85,B 0,C 180,E1 19212.904,E2 19212.904} C_VEL
LIN {X 0,Y 433.491,Z 668.347,A -85,B 0,C 180,E1 19210.866,E2 19210.866} C_VEL
LIN {X 0,Y 432.897,Z 663.602,A -85,B 0,C 180,E1 19210.244,E2 19210.244} C_VEL
LIN {X 0,Y 433.086,Z 649.903,A -85,B 0,C 180,E1 19208.561,E2 19208.561} C_VEL
LIN {X 0,Y 428.275,Z 631.652,A -85,B 0,C 180,E1 19205.956,E2 19205.956} C_VEL
LIN {X 0,Y 425.286,Z 621.442,A -85,B 0,C 180,E1 19204.424,E2 19204.424} C_VEL
LIN {X 0,Y 425.263,Z 621.259,A -85,B 0,C 180,E1 19200.678,E2 19200.678} C_VEL
LIN {X 0,Y 425.292,Z 621.255,A -85,B 0,C 180,E1 19196.984,E2 19196.984} C_VEL
LIN {X 0,Y 425.317,Z 621.237,A -85,B 0,C 180,E1 19193.116,E2 19193.116} C_VEL
LIN {X 0,Y 425.297,Z 621.23,A -85,B 0,C 180,E1 19189.359,E2 19189.359} C_VEL
LIN {X 0,Y 425.333,Z 621.561,A -85,B 0,C 180,E1 19188.525,E2 19188.525} C_VEL
LIN {X 0,Y 430.305,Z 638.377,A -85,B 0,C 180,E1 19185.355,E2 19185.355} C_VEL
LIN {X 0,Y 434.653,Z 654.945,A -85,B 0,C 180,E1 19182.421,E2 19182.421} C_VEL
LIN {X 0,Y 432.6,Z 680.737,A -85,B 0,C 180,E1 19178.641,E2 19178.641} C_VEL
LIN {X 0,Y 431.631,Z 694.711,A -85,B 0,C 180,E1 19176.651,E2 19176.651} C_VEL
LIN {X 0,Y 436.425,Z 719.156,A -85,B 0,C 180,E1 19175.887,E2 19175.887} C_VEL
LIN {X 0,Y 434.386,Z 843.848,A -85,B 0,C 180,E1 19173.737,E2 19173.737} C_VEL
LIN {X 0,Y 433.899,Z 860.973,A -85,B 0,C 180,E1 19173.183,E2 19173.183} C_VEL
LIN {X 0,Y 433.205,Z 876.45,A -85,B 0,C 180,E1 19172.448,E2 19172.448} C_VEL
LIN {X 0,Y 432.246,Z 891.772,A -85,B 0,C 180,E1 19171.458,E2 19171.458} C_VEL
LIN {X 0,Y 431.102,Z 906.78,A -85,B 0,C 180,E1 19170.2,E2 19170.2} C_VEL
LIN {X 0,Y 429.972,Z 919.913,A -85,B 0,C 180,E1 19168.801,E2 19168.801} C_VEL
LIN {X 0,Y 428.824,Z 931.98,A -85,B 0,C 180,E1 19167.194,E2 19167.194} C_VEL
LIN {X 0,Y 427.773,Z 942.585,A -85,B 0,C 180,E1 19165.442,E2 19165.442} C_VEL
LIN {X 0,Y 426.863,Z 951.665,A -85,B 0,C 180,E1 19163.545,E2 19163.545} C_VEL
LIN {X 0,Y 426.144,Z 959.304,A -85,B 0,C 180,E1 19161.5,E2 19161.5} C_VEL
LIN {X 0,Y 425.654,Z 965.105,A -85,B 0,C 180,E1 19159.443,E2 19159.443} C_VEL
LIN {X 0,Y 425.322,Z 969.409,A -85,B 0,C 180,E1 19157.234,E2 19157.234} C_VEL
LIN {X 0,Y 425.157,Z 972.123,A -85,B 0,C 180,E1 19154.868,E2 19154.868} C_VEL
LIN {X 0,Y 425.137,Z 972.903,A -85,B 0,C 180,E1 19152.622,E2 19152.622} C_VEL
LIN {X 0,Y 425.268,Z 971.88,A -85,B 0,C 180,E1 19150.211,E2 19150.211} C_VEL
LIN {X 0,Y 425.548,Z 969.32,A -85,B 0,C 180,E1 19148.064,E2 19148.064} C_VEL
LIN {X 0,Y 425.995,Z 964.991,A -85,B 0,C 180,E1 19145.896,E2 19145.896} C_VEL
LIN {X 0,Y 426.685,Z 958.783,A -85,B 0,C 180,E1 19143.712,E2 19143.712} C_VEL
LIN {X 0,Y 427.536,Z 951.618,A -85,B 0,C 180,E1 19141.81,E2 19141.81} C_VEL
LIN {X 0,Y 428.636,Z 942.38,A -85,B 0,C 180,E1 19139.9,E2 19139.9} C_VEL
LIN {X 0,Y 429.934,Z 931.373,A -85,B 0,C 180,E1 19138.087,E2 19138.087} C_VEL
LIN {X 0,Y 431.253,Z 919.346,A -85,B 0,C 180,E1 19136.51,E2 19136.51} C_VEL
LIN {X 0,Y 432.573,Z 906.033,A -85,B 0,C 180,E1 19135.113,E2 19135.113} C_VEL
LIN {X 0,Y 433.836,Z 891.355,A -85,B 0,C 180,E1 19133.894,E2 19133.894} C_VEL
LIN {X 0,Y 434.896,Z 875.926,A -85,B 0,C 180,E1 19132.919,E2 19132.919} C_VEL
LIN {X 0,Y 435.718,Z 859.384,A -85,B 0,C 180,E1 19132.151,E2 19132.151} C_VEL
LIN {X 0,Y 436.178,Z 842.934,A -85,B 0,C 180,E1 19131.651,E2 19131.651} C_VEL
LIN {X 0,Y 438.417,Z 718.238,A -85,B 0,C 180,E1 19129.437,E2 19129.437} C_VEL
LIN {X 0,Y 433.278,Z 695.593,A -85,B 0,C 180,E1 19128.59,E2 19128.59} C_VEL
LIN {X 0,Y 433.554,Z 690.904,A -85,B 0,C 180,E1 19127.953,E2 19127.953} C_VEL
LIN {X 0,Y 436.064,Z 664.274,A -85,B 0,C 180,E1 19123.948,E2 19123.948} C_VEL
LIN {X 0,Y 436.568,Z 658.374,A -85,B 0,C 180,E1 19123.04,E2 19123.04} C_VEL
LIN {X 0,Y 432.614,Z 643.53,A -85,B 0,C 180,E1 19120.153,E2 19120.153} C_VEL
LIN {X 0,Y 428.423,Z 630.276,A -85,B 0,C 180,E1 19117.358,E2 19117.358} C_VEL
LIN {X 0,Y 425.327,Z 621.372,A -85,B 0,C 180,E1 19115.289,E2 19115.289} C_VEL
LIN {X 0,Y 425.319,Z 621.247,A -85,B 0,C 180,E1 19111.422,E2 19111.422} C_VEL
LIN {X 0,Y 425.31,Z 621.256,A -85,B 0,C 180,E1 19107.589,E2 19107.589} C_VEL
LIN {X 0,Y 425.309,Z 621.257,A -85,B 0,C 180,E1 19103.704,E2 19103.704} C_VEL
LIN {X 0,Y 425.315,Z 621.255,A -85,B 0,C 180,E1 19099.891,E2 19099.891} C_VEL
LIN {X 0,Y 425.317,Z 621.255,A -85,B 0,C 180,E1 19095.965,E2 19095.965} C_VEL
LIN {X 0,Y 425.313,Z 621.257,A -85,B 0,C 180,E1 19092.051,E2 19092.051} C_VEL
LIN {X 0,Y 425.316,Z 621.254,A -85,B 0,C 180,E1 19088.109,E2 19088.109} C_VEL
LIN {X 0,Y 425.31,Z 621.25,A -85,B 0,C 180,E1 19084.315,E2 19084.315} C_VEL
LIN {X 0,Y 425.3,Z 621.24,A -85,B 0,C 180,E1 19080.539,E2 19080.539} C_VEL
LIN {X 0,Y 425.304,Z 621.243,A -85,B 0,C 180,E1 19076.766,E2 19076.766} C_VEL
LIN {X 0,Y 425.323,Z 621.252,A -85,B 0,C 180,E1 19072.843,E2 19072.843} C_VEL
LIN {X 0,Y 425.314,Z 621.252,A -85,B 0,C 180,E1 19068.886,E2 19068.886} C_VEL
LIN {X 0,Y 425.316,Z 621.243,A -85,B 0,C 180,E1 19065.014,E2 19065.014} C_VEL
LIN {X 0,Y 425.311,Z 621.237,A -85,B 0,C 180,E1 19061.212,E2 19061.212} C_VEL
LIN {X 0,Y 425.298,Z 621.245,A -85,B 0,C 180,E1 19057.468,E2 19057.468} C_VEL
LIN {X 0,Y 425.299,Z 621.249,A -85,B 0,C 180,E1 19053.6,E2 19053.6} C_VEL
LIN {X 0,Y 425.314,Z 621.249,A -85,B 0,C 180,E1 19049.796,E2 19049.796} C_VEL
LIN {X 0,Y 425.318,Z 621.25,A -85,B 0,C 180,E1 19045.979,E2 19045.979} C_VEL
LIN {X 0,Y 425.32,Z 621.246,A -85,B 0,C 180,E1 19042.152,E2 19042.152} C_VEL
LIN {X 0,Y 425.303,Z 621.252,A -85,B 0,C 180,E1 19038.382,E2 19038.382} C_VEL
LIN {X 0,Y 425.293,Z 621.256,A -85,B 0,C 180,E1 19034.574,E2 19034.574} C_VEL
LIN {X 0,Y 425.362,Z 621.55,A -85,B 0,C 180,E1 19033.42,E2 19033.42} C_VEL
LIN {X 0,Y 431.375,Z 636.607,A -85,B 0,C 180,E1 19030.718,E2 19030.718} C_VEL
LIN {X 0,Y 436.984,Z 651.884,A -85,B 0,C 180,E1 19028.297,E2 19028.297} C_VEL
LIN {X 0,Y 441.314,Z 665.771,A -85,B 0,C 180,E1 19026.332,E2 19026.332} C_VEL
LIN {X 0,Y 437.365,Z 705.608,A -85,B 0,C 180,E1 19022.418,E2 19022.418} C_VEL
LIN {X 0,Y 437.304,Z 708.639,A -85,B 0,C 180,E1 19022.188,E2 19022.188} C_VEL
LIN {X 0,Y 440.819,Z 736.742,A -85,B 0,C 180,E1 19021.407,E2 19021.407} C_VEL
LIN {X 0,Y 437.492,Z 919.912,A -85,B 0,C 180,E1 19018.285,E2 19018.285} C_VEL
LIN {X 0,Y 436.519,Z 939.114,A -85,B 0,C 180,E1 19017.731,E2 19017.731} C_VEL
LIN {X 0,Y 435.313,Z 957.183,A -85,B 0,C 180,E1 19016.978,E2 19016.978} C_VEL
LIN {X 0,Y 433.854,Z 975.362,A -85,B 0,C 180,E1 19015.968,E2 19015.968} C_VEL
LIN {X 0,Y 432.293,Z 992.646,A -85,B 0,C 180,E1 19014.748,E2 19014.748} C_VEL
LIN {X 0,Y 430.704,Z 1009.095,A -85,B 0,C 180,E1 19013.316,E2 19013.316} C_VEL
LIN {X 0,Y 429.225,Z 1024.079,A -85,B 0,C 180,E1 19011.739,E2 19011.739} C_VEL
LIN {X 0,Y 427.8,Z 1038.8,A -85,B 0,C 180,E1 19009.88,E2 19009.88} C_VEL
LIN {X 0,Y 426.589,Z 1052.017,A -85,B 0,C 180,E1 19007.881,E2 19007.881} C_VEL
LIN {X 0,Y 425.677,Z 1063.448,A -85,B 0,C 180,E1 19005.811,E2 19005.811} C_VEL
LIN {X 0,Y 424.991,Z 1073.549,A -85,B 0,C 180,E1 19003.607,E2 19003.607} C_VEL
LIN {X 0,Y 424.568,Z 1082.258,A -85,B 0,C 180,E1 19001.272,E2 19001.272} C_VEL
LIN {X 0,Y 424.342,Z 1089.46,A -85,B 0,C 180,E1 18998.81,E2 18998.81} C_VEL
LIN {X 0,Y 424.274,Z 1094.787,A -85,B 0,C 180,E1 18996.359,E2 18996.359} C_VEL
LIN {X 0,Y 424.299,Z 1098.346,A -85,B 0,C 180,E1 18993.918,E2 18993.918} C_VEL
LIN {X 0,Y 424.337,Z 1100.189,A -85,B 0,C 180,E1 18991.485,E2 18991.485} C_VEL
LIN {X 0,Y 424.341,Z 1100.376,A -85,B 0,C 180,E1 18989.055,E2 18989.055} C_VEL
LIN {X 0,Y 424.307,Z 1098.916,A -85,B 0,C 180,E1 18986.622,E2 18986.622} C_VEL
LIN {X 0,Y 424.274,Z 1095.785,A -85,B 0,C 180,E1 18984.184,E2 18984.184} C_VEL
LIN {X 0,Y 424.303,Z 1090.913,A -85,B 0,C 180,E1 18981.735,E2 18981.735} C_VEL
LIN {X 0,Y 424.489,Z 1084.199,A -85,B 0,C 180,E1 18979.276,E2 18979.276} C_VEL
LIN {X 0,Y 424.883,Z 1075.468,A -85,B 0,C 180,E1 18976.805,E2 18976.805} C_VEL
LIN {X 0,Y 425.573,Z 1065.125,A -85,B 0,C 180,E1 18974.464,E2 18974.464} C_VEL
LIN {X 0,Y 426.529,Z 1053.207,A -85,B 0,C 180,E1 18972.257,E2 18972.257} C_VEL
LIN {X 0,Y 427.727,Z 1040.197,A -85,B 0,C 180,E1 18970.258,E2 18970.258} C_VEL
LIN {X 0,Y 429.134,Z 1025.686,A -85,B 0,C 180,E1 18968.399,E2 18968.399} C_VEL
LIN {X 0,Y 430.661,Z 1010.208,A -85,B 0,C 180,E1 18966.753,E2 18966.753} C_VEL
LIN {X 0,Y 432.238,Z 993.804,A -85,B 0,C 180,E1 18965.32,E2 18965.32} C_VEL
LIN {X 0,Y 433.777,Z 976.563,A -85,B 0,C 180,E1 18964.1,E2 18964.1} C_VEL
LIN {X 0,Y 435.204,Z 958.442,A -85,B 0,C 180,E1 18963.089,E2 18963.089} C_VEL
LIN {X 0,Y 436.442,Z 939.629,A -85,B 0,C 180,E1 18962.304,E2 18962.304} C_VEL
LIN {X 0,Y 437.39,Z 920.179,A -85,B 0,C 180,E1 18961.748,E2 18961.748} C_VEL
LIN {X 0,Y 440.347,Z 733.926,A -85,B 0,C 180,E1 18958.614,E2 18958.614} C_VEL
LIN {X 0,Y 436.874,Z 707.653,A -85,B 0,C 180,E1 18957.89,E2 18957.89} C_VEL
LIN {X 0,Y 440.334,Z 667.219,A -85,B 0,C 180,E1 18954.057,E2 18954.057} C_VEL
LIN {X 0,Y 440.352,Z 663.907,A -85,B 0,C 180,E1 18953.712,E2 18953.712} C_VEL
LIN {X 0,Y 432.751,Z 641.823,A -85,B 0,C 180,E1 18950.715,E2 18950.715} C_VEL
LIN {X 0,Y 425.365,Z 621.654,A -85,B 0,C 180,E1 18947.712,E2 18947.712} C_VEL
LIN {X 0,Y 425.314,Z 621.26,A -85,B 0,C 180,E1 18946.98,E2 18946.98} C_VEL
LIN {X 0,Y 425.309,Z 621.254,A -85,B 0,C 180,E1 18943.166,E2 18943.166} C_VEL
LIN {X 0,Y 425.31,Z 621.254,A -85,B 0,C 180,E1 18939.335,E2 18939.335} C_VEL
LIN {X 0,Y 425.317,Z 621.255,A -85,B 0,C 180,E1 18935.497,E2 18935.497} C_VEL
LIN {X 0,Y 425.311,Z 621.255,A -85,B 0,C 180,E1 18931.617,E2 18931.617} C_VEL
LIN {X 0,Y 425.299,Z 621.256,A -85,B 0,C 180,E1 18927.875,E2 18927.875} C_VEL
LIN {X 0,Y 425.298,Z 621.261,A -85,B 0,C 180,E1 18923.999,E2 18923.999} C_VEL
LIN {X 0,Y 425.311,Z 621.258,A -85,B 0,C 180,E1 18920.217,E2 18920.217} C_VEL
LIN {X 0,Y 425.322,Z 621.258,A -85,B 0,C 180,E1 18916.385,E2 18916.385} C_VEL
LIN {X 0,Y 425.309,Z 621.26,A -85,B 0,C 180,E1 18912.629,E2 18912.629} C_VEL
LIN {X 0,Y 425.372,Z 621.628,A -85,B 0,C 180,E1 18912.194,E2 18912.194} C_VEL
LIN {X 0,Y 430.506,Z 636.234,A -85,B 0,C 180,E1 18910.017,E2 18910.017} C_VEL
LIN {X 0,Y 434.68,Z 651.211,A -85,B 0,C 180,E1 18907.933,E2 18907.933} C_VEL
LIN {X 0,Y 434.959,Z 655.632,A -85,B 0,C 180,E1 18907.396,E2 18907.396} C_VEL
LIN {X 0,Y 434.539,Z 686.014,A -85,B 0,C 180,E1 18903.892,E2 18903.892} C_VEL
LIN {X 0,Y 434.039,Z 716.181,A -85,B 0,C 180,E1 18900.359,E2 18900.359} C_VEL
LIN {X 0,Y 434.299,Z 720.237,A -85,B 0,C 180,E1 18900.253,E2 18900.253} C_VEL
LIN {X 0,Y 431.779,Z 847.368,A -85,B 0,C 180,E1 18897.81,E2 18897.81} C_VEL
LIN {X 0,Y 431.705,Z 863.961,A -85,B 0,C 180,E1 18897.353,E2 18897.353} C_VEL
LIN {X 0,Y 431.345,Z 880.458,A -85,B 0,C 180,E1 18896.63,E2 18896.63} C_VEL
LIN {X 0,Y 430.799,Z 895.001,A -85,B 0,C 180,E1 18895.74,E2 18895.74} C_VEL
LIN {X 0,Y 430.064,Z 909.26,A -85,B 0,C 180,E1 18894.597,E2 18894.597} C_VEL
LIN {X 0,Y 429.277,Z 921.823,A -85,B 0,C 180,E1 18893.312,E2 18893.312} C_VEL
LIN {X 0,Y 428.384,Z 934.05,A -85,B 0,C 180,E1 18891.743,E2 18891.743} C_VEL
LIN {X 0,Y 427.607,Z 943.824,A -85,B 0,C 180,E1 18890.172,E2 18890.172} C_VEL
LIN {X 0,Y 426.82,Z 953.302,A -85,B 0,C 180,E1 18888.24,E2 18888.24} C_VEL
LIN {X 0,Y 426.215,Z 960.605,A -85,B 0,C 180,E1 18886.294,E2 18886.294} C_VEL
LIN {X 0,Y 425.743,Z 966.422,A -85,B 0,C 180,E1 18884.191,E2 18884.191} C_VEL
LIN {X 0,Y 425.415,Z 970.332,A -85,B 0,C 180,E1 18882.067,E2 18882.067} C_VEL
LIN {X 0,Y 425.229,Z 972.498,A -85,B 0,C 180,E1 18879.922,E2 18879.922} C_VEL
LIN {X 0,Y 425.146,Z 972.909,A -85,B 0,C 180,E1 18877.75,E2 18877.75} C_VEL
LIN {X 0,Y 425.156,Z 971.509,A -85,B 0,C 180,E1 18875.524,E2 18875.524} C_VEL
LIN {X 0,Y 425.27,Z 968.549,A -85,B 0,C 180,E1 18873.467,E2 18873.467} C_VEL
LIN {X 0,Y 425.541,Z 963.335,A -85,B 0,C 180,E1 18871.205,E2 18871.205} C_VEL
LIN {X 0,Y 425.928,Z 956.856,A -85,B 0,C 180,E1 18869.219,E2 18869.219} C_VEL
LIN {X 0,Y 426.493,Z 948.256,A -85,B 0,C 180,E1 18867.21,E2 18867.21} C_VEL
LIN {X 0,Y 427.169,Z 938.372,A -85,B 0,C 180,E1 18865.416,E2 18865.416} C_VEL
LIN {X 0,Y 427.952,Z 927.019,A -85,B 0,C 180,E1 18863.764,E2 18863.764} C_VEL
LIN {X 0,Y 428.735,Z 914.703,A -85,B 0,C 180,E1 18862.337,E2 18862.337} C_VEL
LIN {X 0,Y 429.526,Z 900.639,A -85,B 0,C 180,E1 18861.032,E2 18861.032} C_VEL
LIN {X 0,Y 430.189,Z 886.105,A -85,B 0,C 180,E1 18859.991,E2 18859.991} C_VEL
LIN {X 0,Y 430.737,Z 870.636,A -85,B 0,C 180,E1 18859.15,E2 18859.15} C_VEL
LIN {X 0,Y 431.057,Z 854.008,A -85,B 0,C 180,E1 18858.528,E2 18858.528} C_VEL
LIN {X 0,Y 431.175,Z 835.403,A -85,B 0,C 180,E1 18858.115,E2 18858.115} C_VEL
LIN {X 0,Y 433.024,Z 715.367,A -85,B 0,C 180,E1 18855.92,E2 18855.92} C_VEL
LIN {X 0,Y 431.692,Z 708.031,A -85,B 0,C 180,E1 18855.686,E2 18855.686} C_VEL
LIN {X 0,Y 432.513,Z 678.112,A -85,B 0,C 180,E1 18852.019,E2 18852.019} C_VEL
LIN {X 0,Y 432.897,Z 663.602,A -85,B 0,C 180,E1 18850.244,E2 18850.244} C_VEL
LIN {X 0,Y 432.21,Z 659.002,A -85,B 0,C 180,E1 18849.616,E2 18849.616} C_VEL
LIN {X 0,Y 429.2,Z 652.81,A -85,B 0,C 180,E1 18848.635,E2 18848.635} C_VEL
LIN {X 0,Y 423.619,Z 643.438,A -85,B 0,C 180,E1 18847.07,E2 18847.07} C_VEL
LIN {X 0,Y 422.828,Z 641.192,A -85,B 0,C 180,E1 18846.739,E2 18846.739} C_VEL
LIN {X 0,Y 417.373,Z 622.402,A -85,B 0,C 180,E1 18843.93,E2 18843.93} C_VEL
LIN {X 0,Y 417.329,Z 622.248,A -85,B 0,C 180,E1 18840.208,E2 18840.208} C_VEL
LIN {X 0,Y 417.325,Z 622.237,A -85,B 0,C 180,E1 18836.355,E2 18836.355} C_VEL
LIN {X 0,Y 417.335,Z 622.245,A -85,B 0,C 180,E1 18832.541,E2 18832.541} C_VEL
LIN {X 0,Y 417.409,Z 622.487,A -85,B 0,C 180,E1 18829.147,E2 18829.147} C_VEL
LIN {X 0,Y 422.718,Z 640.401,A -85,B 0,C 180,E1 18825.701,E2 18825.701} C_VEL
LIN {X 0,Y 427.154,Z 657.332,A -85,B 0,C 180,E1 18822.642,E2 18822.642} C_VEL
LIN {X 0,Y 424.926,Z 684.201,A -85,B 0,C 180,E1 18818.662,E2 18818.662} C_VEL
LIN {X 0,Y 424.139,Z 694.684,A -85,B 0,C 180,E1 18817.144,E2 18817.144} C_VEL
LIN {X 0,Y 425.951,Z 703.943,A -85,B 0,C 180,E1 18816.813,E2 18816.813} C_VEL
LIN {X 0,Y 429.153,Z 720.475,A -85,B 0,C 180,E1 18816.314,E2 18816.314} C_VEL
LIN {X 0,Y 427.016,Z 844.544,A -85,B 0,C 180,E1 18814.142,E2 18814.142} C_VEL
LIN {X 0,Y 426.506,Z 861.685,A -85,B 0,C 180,E1 18813.579,E2 18813.579} C_VEL
LIN {X 0,Y 425.773,Z 877.266,A -85,B 0,C 180,E1 18812.827,E2 18812.827} C_VEL
LIN {X 0,Y 424.767,Z 892.606,A -85,B 0,C 180,E1 18811.821,E2 18811.821} C_VEL
LIN {X 0,Y 423.563,Z 907.636,A -85,B 0,C 180,E1 18810.541,E2 18810.541} C_VEL
LIN {X 0,Y 422.371,Z 920.802,A -85,B 0,C 180,E1 18809.119,E2 18809.119} C_VEL
LIN {X 0,Y 421.205,Z 932.439,A -85,B 0,C 180,E1 18807.551,E2 18807.551} C_VEL
LIN {X 0,Y 420.081,Z 943.151,A -85,B 0,C 180,E1 18805.769,E2 18805.769} C_VEL
LIN {X 0,Y 419.108,Z 952.371,A -85,B 0,C 180,E1 18803.837,E2 18803.837} C_VEL
LIN {X 0,Y 418.316,Z 960.249,A -85,B 0,C 180,E1 18801.709,E2 18801.709} C_VEL
LIN {X 0,Y 417.769,Z 966.331,A -85,B 0,C 180,E1 18799.52,E2 18799.52} C_VEL
LIN {X 0,Y 417.418,Z 970.619,A -85,B 0,C 180,E1 18797.269,E2 18797.269} C_VEL
LIN {X 0,Y 417.247,Z 973.243,A -85,B 0,C 180,E1 18794.956,E2 18794.956} C_VEL
LIN {X 0,Y 417.227,Z 974.113,A -85,B 0,C 180,E1 18792.713,E2 18792.713} C_VEL
LIN {X 0,Y 417.356,Z 973.221,A -85,B 0,C 180,E1 18790.308,E2 18790.308} C_VEL
LIN {X 0,Y 417.658,Z 970.739,A -85,B 0,C 180,E1 18788.071,E2 18788.071} C_VEL
LIN {X 0,Y 418.137,Z 966.571,A -85,B 0,C 180,E1 18785.865,E2 18785.865} C_VEL
LIN {X 0,Y 418.866,Z 960.493,A -85,B 0,C 180,E1 18783.641,E2 18783.641} C_VEL
LIN {X 0,Y 419.845,Z 952.891,A -85,B 0,C 180,E1 18781.556,E2 18781.556} C_VEL
LIN {X 0,Y 421.025,Z 943.696,A -85,B 0,C 180,E1 18779.613,E2 18779.613} C_VEL
LIN {X 0,Y 422.436,Z 932.566,A -85,B 0,C 180,E1 18777.742,E2 18777.742} C_VEL
LIN {X 0,Y 423.846,Z 920.584,A -85,B 0,C 180,E1 18776.138,E2 18776.138} C_VEL
LIN {X 0,Y 425.314,Z 906.745,A -85,B 0,C 180,E1 18774.663,E2 18774.663} C_VEL
LIN {X 0,Y 426.611,Z 892.562,A -85,B 0,C 180,E1 18773.466,E2 18773.466} C_VEL
LIN {X 0,Y 427.723,Z 877.408,A -85,B 0,C 180,E1 18772.486,E2 18772.486} C_VEL
LIN {X 0,Y 428.606,Z 860.763,A -85,B 0,C 180,E1 18771.694,E2 18771.694} C_VEL
LIN {X 0,Y 429.115,Z 844.286,A -85,B 0,C 180,E1 18771.174,E2 18771.174} C_VEL
LIN {X 0,Y 431.515,Z 719.624,A -85,B 0,C 180,E1 18768.919,E2 18768.919} C_VEL
LIN {X 0,Y 426.051,Z 695.415,A -85,B 0,C 180,E1 18767.968,E2 18767.968} C_VEL
LIN {X 0,Y 428.406,Z 670.616,A -85,B 0,C 180,E1 18764.233,E2 18764.233} C_VEL
LIN {X 0,Y 429.376,Z 661.501,A -85,B 0,C 180,E1 18762.818,E2 18762.818} C_VEL
LIN {X 0,Y 425.503,Z 646.802,A -85,B 0,C 180,E1 18759.904,E2 18759.904} C_VEL
LIN {X 0,Y 421.293,Z 633.656,A -85,B 0,C 180,E1 18757.073,E2 18757.073} C_VEL
LIN {X 0,Y 417.391,Z 622.359,A -85,B 0,C 180,E1 18754.38,E2 18754.38} C_VEL
LIN {X 0,Y 417.383,Z 622.242,A -85,B 0,C 180,E1 18750.414,E2 18750.414} C_VEL
LIN {X 0,Y 417.375,Z 622.241,A -85,B 0,C 180,E1 18746.461,E2 18746.461} C_VEL
LIN {X 0,Y 417.372,Z 622.235,A -85,B 0,C 180,E1 18742.538,E2 18742.538} C_VEL
LIN {X 0,Y 417.375,Z 622.232,A -85,B 0,C 180,E1 18738.724,E2 18738.724} C_VEL
LIN {X 0,Y 417.372,Z 622.231,A -85,B 0,C 180,E1 18734.853,E2 18734.853} C_VEL
LIN {X 0,Y 417.365,Z 622.236,A -85,B 0,C 180,E1 18731.049,E2 18731.049} C_VEL
LIN {X 0,Y 417.371,Z 622.242,A -85,B 0,C 180,E1 18727.156,E2 18727.156} C_VEL
LIN {X 0,Y 417.374,Z 622.246,A -85,B 0,C 180,E1 18723.296,E2 18723.296} C_VEL
LIN {X 0,Y 417.375,Z 622.234,A -85,B 0,C 180,E1 18719.451,E2 18719.451} C_VEL
LIN {X 0,Y 417.374,Z 622.223,A -85,B 0,C 180,E1 18715.604,E2 18715.604} C_VEL
LIN {X 0,Y 417.374,Z 622.231,A -85,B 0,C 180,E1 18711.736,E2 18711.736} C_VEL
LIN {X 0,Y 417.365,Z 622.241,A -85,B 0,C 180,E1 18707.801,E2 18707.801} C_VEL
LIN {X 0,Y 417.362,Z 622.248,A -85,B 0,C 180,E1 18704.008,E2 18704.008} C_VEL
LIN {X 0,Y 417.369,Z 622.236,A -85,B 0,C 180,E1 18700.112,E2 18700.112} C_VEL
LIN {X 0,Y 417.378,Z 622.23,A -85,B 0,C 180,E1 18696.268,E2 18696.268} C_VEL
LIN {X 0,Y 417.379,Z 622.23,A -85,B 0,C 180,E1 18692.419,E2 18692.419} C_VEL
LIN {X 0,Y 417.38,Z 622.23,A -85,B 0,C 180,E1 18688.518,E2 18688.518} C_VEL
LIN {X 0,Y 417.363,Z 622.236,A -85,B 0,C 180,E1 18684.736,E2 18684.736} C_VEL
LIN {X 0,Y 417.355,Z 622.245,A -85,B 0,C 180,E1 18680.914,E2 18680.914} C_VEL
LIN {X 0,Y 417.364,Z 622.243,A -85,B 0,C 180,E1 18677.128,E2 18677.128} C_VEL
LIN {X 0,Y 417.398,Z 622.517,A -85,B 0,C 180,E1 18674.363,E2 18674.363} C_VEL
LIN {X 0,Y 423.167,Z 636.484,A -85,B 0,C 180,E1 18671.7,E2 18671.7} C_VEL
LIN {X 0,Y 429.281,Z 652.955,A -85,B 0,C 180,E1 18668.966,E2 18668.966} C_VEL
LIN {X 0,Y 434.179,Z 668.399,A -85,B 0,C 180,E1 18666.691,E2 18666.691} C_VEL
LIN {X 0,Y 430.149,Z 706.486,A -85,B 0,C 180,E1 18662.871,E2 18662.871} C_VEL
LIN {X 0,Y 430.275,Z 709.296,A -85,B 0,C 180,E1 18662.71,E2 18662.71} C_VEL
LIN {X 0,Y 433.782,Z 737.717,A -85,B 0,C 180,E1 18661.896,E2 18661.896} C_VEL
LIN {X 0,Y 430.281,Z 919.016,A -85,B 0,C 180,E1 18658.756,E2 18658.756} C_VEL
LIN {X 0,Y 429.248,Z 938.283,A -85,B 0,C 180,E1 18658.193,E2 18658.193} C_VEL
LIN {X 0,Y 427.938,Z 956.756,A -85,B 0,C 180,E1 18657.405,E2 18657.405} C_VEL
LIN {X 0,Y 426.42,Z 974.465,A -85,B 0,C 180,E1 18656.401,E2 18656.401} C_VEL
LIN {X 0,Y 424.746,Z 991.914,A -85,B 0,C 180,E1 18655.144,E2 18655.144} C_VEL
LIN {X 0,Y 423.069,Z 1008.294,A -85,B 0,C 180,E1 18653.688,E2 18653.688} C_VEL
LIN {X 0,Y 421.438,Z 1023.812,A -85,B 0,C 180,E1 18652.015,E2 18652.015} C_VEL
LIN {X 0,Y 419.943,Z 1038.373,A -85,B 0,C 180,E1 18650.123,E2 18650.123} C_VEL
LIN {X 0,Y 418.678,Z 1051.445,A -85,B 0,C 180,E1 18648.086,E2 18648.086} C_VEL
LIN {X 0,Y 417.651,Z 1063.797,A -85,B 0,C 180,E1 18645.764,E2 18645.764} C_VEL
LIN {X 0,Y 416.956,Z 1073.889,A -85,B 0,C 180,E1 18643.45,E2 18643.45} C_VEL
LIN {X 0,Y 416.549,Z 1082.721,A -85,B 0,C 180,E1 18640.931,E2 18640.931} C_VEL
LIN {X 0,Y 416.368,Z 1089.522,A -85,B 0,C 180,E1 18638.423,E2 18638.423} C_VEL
LIN {X 0,Y 416.349,Z 1094.464,A -85,B 0,C 180,E1 18635.927,E2 18635.927} C_VEL
LIN {X 0,Y 416.394,Z 1097.658,A -85,B 0,C 180,E1 18633.441,E2 18633.441} C_VEL
LIN {X 0,Y 416.431,Z 1099.171,A -85,B 0,C 180,E1 18630.963,E2 18630.963} C_VEL
LIN {X 0,Y 416.419,Z 1099.097,A -85,B 0,C 180,E1 18628.624,E2 18628.624} C_VEL
LIN {X 0,Y 416.368,Z 1097.36,A -85,B 0,C 180,E1 18626.144,E2 18626.144} C_VEL
LIN {X 0,Y 416.322,Z 1093.917,A -85,B 0,C 180,E1 18623.657,E2 18623.657} C_VEL
LIN {X 0,Y 416.367,Z 1088.718,A -85,B 0,C 180,E1 18621.159,E2 18621.159} C_VEL
LIN {X 0,Y 416.567,Z 1082.08,A -85,B 0,C 180,E1 18618.789,E2 18618.789} C_VEL
LIN {X 0,Y 416.983,Z 1073.621,A -85,B 0,C 180,E1 18616.409,E2 18616.409} C_VEL
LIN {X 0,Y 417.678,Z 1063.775,A -85,B 0,C 180,E1 18614.163,E2 18614.163} C_VEL
LIN {X 0,Y 418.687,Z 1051.803,A -85,B 0,C 180,E1 18611.913,E2 18611.913} C_VEL
LIN {X 0,Y 419.96,Z 1038.713,A -85,B 0,C 180,E1 18609.877,E2 18609.877} C_VEL
LIN {X 0,Y 421.458,Z 1024.077,A -85,B 0,C 180,E1 18607.985,E2 18607.985} C_VEL
LIN {X 0,Y 423.083,Z 1008.439,A -85,B 0,C 180,E1 18606.312,E2 18606.312} C_VEL
LIN {X 0,Y 424.75,Z 991.87,A -85,B 0,C 180,E1 18604.855,E2 18604.855} C_VEL
LIN {X 0,Y 426.389,Z 974.266,A -85,B 0,C 180,E1 18603.607,E2 18603.607} C_VEL
LIN {X 0,Y 427.901,Z 955.935,A -85,B 0,C 180,E1 18602.592,E2 18602.592} C_VEL
LIN {X 0,Y 429.173,Z 936.75,A -85,B 0,C 180,E1 18601.807,E2 18601.807} C_VEL
LIN {X 0,Y 430.114,Z 917.068,A -85,B 0,C 180,E1 18601.271,E2 18601.271} C_VEL
LIN {X 0,Y 433.134,Z 735.032,A -85,B 0,C 180,E1 18598.174,E2 18598.174} C_VEL
LIN {X 0,Y 429.535,Z 707.694,A -85,B 0,C 180,E1 18597.421,E2 18597.421} C_VEL
LIN {X 0,Y 432.994,Z 669.795,A -85,B 0,C 180,E1 18593.761,E2 18593.761} C_VEL
LIN {X 0,Y 433.073,Z 666.724,A -85,B 0,C 180,E1 18593.44,E2 18593.44} C_VEL
LIN {X 0,Y 425.348,Z 644.265,A -85,B 0,C 180,E1 18590.34,E2 18590.34} C_VEL
LIN {X 0,Y 418.226,Z 625.001,A -85,B 0,C 180,E1 18587.42,E2 18587.42} C_VEL
LIN {X 0,Y 417.394,Z 622.385,A -85,B 0,C 180,E1 18586.938,E2 18586.938} C_VEL
LIN {X 0,Y 417.373,Z 622.244,A -85,B 0,C 180,E1 18583.058,E2 18583.058} C_VEL
LIN {X 0,Y 417.371,Z 622.242,A -85,B 0,C 180,E1 18579.23,E2 18579.23} C_VEL
LIN {X 0,Y 417.378,Z 622.245,A -85,B 0,C 180,E1 18575.431,E2 18575.431} C_VEL
LIN {X 0,Y 417.373,Z 622.244,A -85,B 0,C 180,E1 18571.644,E2 18571.644} C_VEL
LIN {X 0,Y 417.36,Z 622.245,A -85,B 0,C 180,E1 18567.85,E2 18567.85} C_VEL
LIN {X 0,Y 417.36,Z 622.249,A -85,B 0,C 180,E1 18564.033,E2 18564.033} C_VEL
LIN {X 0,Y 417.37,Z 622.247,A -85,B 0,C 180,E1 18560.18,E2 18560.18} C_VEL
LIN {X 0,Y 417.379,Z 622.248,A -85,B 0,C 180,E1 18556.277,E2 18556.277} C_VEL
LIN {X 0,Y 417.384,Z 622.508,A -85,B 0,C 180,E1 18552.975,E2 18552.975} C_VEL
LIN {X 0,Y 422.215,Z 635.476,A -85,B 0,C 180,E1 18550.92,E2 18550.92} C_VEL
LIN {X 0,Y 426.408,Z 649.46,A -85,B 0,C 180,E1 18548.903,E2 18548.903} C_VEL
LIN {X 0,Y 427.899,Z 656.135,A -85,B 0,C 180,E1 18547.992,E2 18547.992} C_VEL
LIN {X 0,Y 427.346,Z 689.664,A -85,B 0,C 180,E1 18544.092,E2 18544.092} C_VEL
LIN {X 0,Y 426.808,Z 717.497,A -85,B 0,C 180,E1 18540.805,E2 18540.805} C_VEL
LIN {X 0,Y 427.075,Z 721.394,A -85,B 0,C 180,E1 18540.698,E2 18540.698} C_VEL
LIN {X 0,Y 424.355,Z 850.523,A -85,B 0,C 180,E1 18538.143,E2 18538.143} C_VEL
LIN {X 0,Y 424.231,Z 866.795,A -85,B 0,C 180,E1 18537.657,E2 18537.657} C_VEL
LIN {X 0,Y 423.868,Z 882.183,A -85,B 0,C 180,E1 18536.957,E2 18536.957} C_VEL
LIN {X 0,Y 423.304,Z 896.358,A -85,B 0,C 180,E1 18536.072,E2 18536.072} C_VEL
LIN {X 0,Y 422.528,Z 910.623,A -85,B 0,C 180,E1 18534.909,E2 18534.909} C_VEL
LIN {X 0,Y 421.694,Z 923.194,A -85,B 0,C 180,E1 18533.601,E2 18533.601} C_VEL
LIN {X 0,Y 420.778,Z 934.886,A -85,B 0,C 180,E1 18532.078,E2 18532.078} C_VEL
LIN {X 0,Y 419.906,Z 945.153,A -85,B 0,C 180,E1 18530.405,E2 18530.405} C_VEL
LIN {X 0,Y 419.06,Z 954.62,A -85,B 0,C 180,E1 18528.438,E2 18528.438} C_VEL
LIN {X 0,Y 418.409,Z 961.919,A -85,B 0,C 180,E1 18526.456,E2 18526.456} C_VEL
LIN {X 0,Y 417.896,Z 967.726,A -85,B 0,C 180,E1 18524.314,E2 18524.314} C_VEL
LIN {X 0,Y 417.539,Z 971.616,A -85,B 0,C 180,E1 18522.15,E2 18522.15} C_VEL
LIN {X 0,Y 417.33,Z 973.787,A -85,B 0,C 180,E1 18519.914,E2 18519.914} C_VEL
LIN {X 0,Y 417.236,Z 974.101,A -85,B 0,C 180,E1 18517.67,E2 18517.67} C_VEL
LIN {X 0,Y 417.256,Z 972.567,A -85,B 0,C 180,E1 18515.357,E2 18515.357} C_VEL
LIN {X 0,Y 417.397,Z 969.089,A -85,B 0,C 180,E1 18513.08,E2 18513.08} C_VEL
LIN {X 0,Y 417.687,Z 963.979,A -85,B 0,C 180,E1 18510.925,E2 18510.925} C_VEL
LIN {X 0,Y 418.153,Z 956.68,A -85,B 0,C 180,E1 18508.743,E2 18508.743} C_VEL
LIN {X 0,Y 418.728,Z 948.397,A -85,B 0,C 180,E1 18506.851,E2 18506.851} C_VEL
LIN {X 0,Y 419.501,Z 937.745,A -85,B 0,C 180,E1 18504.941,E2 18504.941} C_VEL
LIN {X 0,Y 420.3,Z 926.463,A -85,B 0,C 180,E1 18503.337,E2 18503.337} C_VEL
LIN {X 0,Y 421.141,Z 913.746,A -85,B 0,C 180,E1 18501.882,E2 18501.882} C_VEL
LIN {X 0,Y 421.926,Z 899.982,A -85,B 0,C 180,E1 18500.632,E2 18500.632} C_VEL
LIN {X 0,Y 422.614,Z 885.262,A -85,B 0,C 180,E1 18499.589,E2 18499.589} C_VEL
LIN {X 0,Y 423.149,Z 869.687,A -85,B 0,C 180,E1 18498.768,E2 18498.768} C_VEL
LIN {X 0,Y 423.476,Z 852.62,A -85,B 0,C 180,E1 18498.148,E2 18498.148} C_VEL
LIN {X 0,Y 423.787,Z 820.037,A -85,B 0,C 180,E1 18497.498,E2 18497.498} C_VEL
LIN {X 0,Y 425.534,Z 716.517,A -85,B 0,C 180,E1 18495.56,E2 18495.56} C_VEL
LIN {X 0,Y 424.187,Z 708.82,A -85,B 0,C 180,E1 18495.29,E2 18495.29} C_VEL
LIN {X 0,Y 425.106,Z 677.736,A -85,B 0,C 180,E1 18491.46,E2 18491.46} C_VEL
LIN {X 0,Y 425.733,Z 652.824,A -85,B 0,C 180,E1 18488.404,E2 18488.404} C_VEL
LIN {X 0,Y 422.828,Z 641.192,A -85,B 0,C 180,E1 18486.739,E2 18486.739} C_VEL
LIN {X 0,Y 420.982,Z 638.128,A -85,B 0,C 180,E1 18486.223,E2 18486.223} C_VEL
LIN {X 0,Y 412.465,Z 631.533,A -85,B 0,C 180,E1 18484.745,E2 18484.745} C_VEL
LIN {X 0,Y 411.155,Z 629.319,A -85,B 0,C 180,E1 18484.363,E2 18484.363} C_VEL
LIN {X 0,Y 409.447,Z 623.395,A -85,B 0,C 180,E1 18483.434,E2 18483.434} C_VEL
LIN {X 0,Y 409.437,Z 623.236,A -85,B 0,C 180,E1 18479.558,E2 18479.558} C_VEL
LIN {X 0,Y 409.41,Z 623.206,A -85,B 0,C 180,E1 18475.687,E2 18475.687} C_VEL
LIN {X 0,Y 409.397,Z 623.24,A -85,B 0,C 180,E1 18471.864,E2 18471.864} C_VEL
LIN {X 0,Y 409.435,Z 623.499,A -85,B 0,C 180,E1 18469.787,E2 18469.787} C_VEL
LIN {X 0,Y 414.375,Z 639.904,A -85,B 0,C 180,E1 18466.543,E2 18466.543} C_VEL
LIN {X 0,Y 418.899,Z 656.849,A -85,B 0,C 180,E1 18463.387,E2 18463.387} C_VEL
LIN {X 0,Y 419.625,Z 660.15,A -85,B 0,C 180,E1 18462.803,E2 18462.803} C_VEL
LIN {X 0,Y 417.248,Z 687.666,A -85,B 0,C 180,E1 18458.683,E2 18458.683} C_VEL
LIN {X 0,Y 416.704,Z 695.087,A -85,B 0,C 180,E1 18457.619,E2 18457.619} C_VEL
LIN {X 0,Y 421.899,Z 721.597,A -85,B 0,C 180,E1 18456.757,E2 18456.757} C_VEL
LIN {X 0,Y 419.656,Z 845.224,A -85,B 0,C 180,E1 18454.557,E2 18454.557} C_VEL
LIN {X 0,Y 419.121,Z 862.402,A -85,B 0,C 180,E1 18453.985,E2 18453.985} C_VEL
LIN {X 0,Y 418.353,Z 878.018,A -85,B 0,C 180,E1 18453.22,E2 18453.22} C_VEL
LIN {X 0,Y 417.302,Z 893.405,A -85,B 0,C 180,E1 18452.197,E2 18452.197} C_VEL
LIN {X 0,Y 416.031,Z 908.546,A -85,B 0,C 180,E1 18450.889,E2 18450.889} C_VEL
LIN {X 0,Y 414.783,Z 921.686,A -85,B 0,C 180,E1 18449.448,E2 18449.448} C_VEL
LIN {X 0,Y 413.504,Z 933.812,A -85,B 0,C 180,E1 18447.783,E2 18447.783} C_VEL
LIN {X 0,Y 412.324,Z 944.475,A -85,B 0,C 180,E1 18445.968,E2 18445.968} C_VEL
LIN {X 0,Y 411.298,Z 953.64,A -85,B 0,C 180,E1 18444,E2 18444} C_VEL
LIN {X 0,Y 410.479,Z 961.345,A -85,B 0,C 180,E1 18441.879,E2 18441.879} C_VEL
LIN {X 0,Y 409.914,Z 967.221,A -85,B 0,C 180,E1 18439.744,E2 18439.744} C_VEL
LIN {X 0,Y 409.533,Z 971.612,A -85,B 0,C 180,E1 18437.45,E2 18437.45} C_VEL
LIN {X 0,Y 409.337,Z 974.404,A -85,B 0,C 180,E1 18434.994,E2 18434.994} C_VEL
LIN {X 0,Y 409.317,Z 975.308,A -85,B 0,C 180,E1 18432.662,E2 18432.662} C_VEL
LIN {X 0,Y 409.454,Z 974.491,A -85,B 0,C 180,E1 18430.307,E2 18430.307} C_VEL
LIN {X 0,Y 409.795,Z 971.948,A -85,B 0,C 180,E1 18427.93,E2 18427.93} C_VEL
LIN {X 0,Y 410.321,Z 967.797,A -85,B 0,C 180,E1 18425.681,E2 18425.681} C_VEL
LIN {X 0,Y 411.112,Z 961.745,A -85,B 0,C 180,E1 18423.417,E2 18423.417} C_VEL
LIN {X 0,Y 412.167,Z 954.183,A -85,B 0,C 180,E1 18421.294,E2 18421.294} C_VEL
LIN {X 0,Y 413.433,Z 945.051,A -85,B 0,C 180,E1 18419.317,E2 18419.317} C_VEL
LIN {X 0,Y 414.955,Z 933.82,A -85,B 0,C 180,E1 18417.39,E2 18417.39} C_VEL
LIN {X 0,Y 416.476,Z 921.725,A -85,B 0,C 180,E1 18415.738,E2 18415.738} C_VEL
LIN {X 0,Y 417.977,Z 908.433,A -85,B 0,C 180,E1 18414.29,E2 18414.29} C_VEL
LIN {X 0,Y 419.351,Z 894.365,A -85,B 0,C 180,E1 18413.07,E2 18413.07} C_VEL
LIN {X 0,Y 420.533,Z 879.623,A -85,B 0,C 180,E1 18412.079,E2 18412.079} C_VEL
LIN {X 0,Y 421.489,Z 863.045,A -85,B 0,C 180,E1 18411.256,E2 18411.256} C_VEL
LIN {X 0,Y 422.086,Z 846.234,A -85,B 0,C 180,E1 18410.693,E2 18410.693} C_VEL
LIN {X 0,Y 424.652,Z 721.007,A -85,B 0,C 180,E1 18408.384,E2 18408.384} C_VEL
LIN {X 0,Y 418.919,Z 695.773,A -85,B 0,C 180,E1 18407.369,E2 18407.369} C_VEL
LIN {X 0,Y 420.152,Z 682.363,A -85,B 0,C 180,E1 18405.361,E2 18405.361} C_VEL
LIN {X 0,Y 422.032,Z 663.993,A -85,B 0,C 180,E1 18402.471,E2 18402.471} C_VEL
LIN {X 0,Y 418.391,Z 650.085,A -85,B 0,C 180,E1 18399.648,E2 18399.648} C_VEL
LIN {X 0,Y 413.849,Z 635.7,A -85,B 0,C 180,E1 18396.466,E2 18396.466} C_VEL
LIN {X 0,Y 409.455,Z 623.34,A -85,B 0,C 180,E1 18393.404,E2 18393.404} C_VEL
LIN {X 0,Y 409.438,Z 623.231,A -85,B 0,C 180,E1 18389.557,E2 18389.557} C_VEL
LIN {X 0,Y 409.431,Z 623.223,A -85,B 0,C 180,E1 18385.611,E2 18385.611} C_VEL
LIN {X 0,Y 409.431,Z 623.224,A -85,B 0,C 180,E1 18381.639,E2 18381.639} C_VEL
LIN {X 0,Y 409.436,Z 623.223,A -85,B 0,C 180,E1 18377.751,E2 18377.751} C_VEL
LIN {X 0,Y 409.438,Z 623.219,A -85,B 0,C 180,E1 18373.847,E2 18373.847} C_VEL
LIN {X 0,Y 409.434,Z 623.216,A -85,B 0,C 180,E1 18369.985,E2 18369.985} C_VEL
LIN {X 0,Y 409.438,Z 623.218,A -85,B 0,C 180,E1 18366.028,E2 18366.028} C_VEL
LIN {X 0,Y 409.437,Z 623.23,A -85,B 0,C 180,E1 18362.1,E2 18362.1} C_VEL
LIN {X 0,Y 409.43,Z 623.233,A -85,B 0,C 180,E1 18358.181,E2 18358.181} C_VEL
LIN {X 0,Y 409.425,Z 623.229,A -85,B 0,C 180,E1 18354.254,E2 18354.254} C_VEL
LIN {X 0,Y 409.422,Z 623.217,A -85,B 0,C 180,E1 18350.299,E2 18350.299} C_VEL
LIN {X 0,Y 409.431,Z 623.215,A -85,B 0,C 180,E1 18346.395,E2 18346.395} C_VEL
LIN {X 0,Y 409.439,Z 623.224,A -85,B 0,C 180,E1 18342.52,E2 18342.52} C_VEL
LIN {X 0,Y 409.443,Z 623.233,A -85,B 0,C 180,E1 18338.513,E2 18338.513} C_VEL
LIN {X 0,Y 409.442,Z 623.234,A -85,B 0,C 180,E1 18334.546,E2 18334.546} C_VEL
LIN {X 0,Y 409.445,Z 623.233,A -85,B 0,C 180,E1 18330.605,E2 18330.605} C_VEL
LIN {X 0,Y 409.435,Z 623.235,A -85,B 0,C 180,E1 18326.634,E2 18326.634} C_VEL
LIN {X 0,Y 409.421,Z 623.23,A -85,B 0,C 180,E1 18322.725,E2 18322.725} C_VEL
LIN {X 0,Y 409.416,Z 623.227,A -85,B 0,C 180,E1 18318.933,E2 18318.933} C_VEL
LIN {X 0,Y 409.467,Z 623.443,A -85,B 0,C 180,E1 18315.377,E2 18315.377} C_VEL
LIN {X 0,Y 412.296,Z 630.364,A -85,B 0,C 180,E1 18313.925,E2 18313.925} C_VEL
LIN {X 0,Y 418.134,Z 644.769,A -85,B 0,C 180,E1 18311.232,E2 18311.232} C_VEL
LIN {X 0,Y 423.728,Z 660.509,A -85,B 0,C 180,E1 18308.643,E2 18308.643} C_VEL
LIN {X 0,Y 427.023,Z 671.664,A -85,B 0,C 180,E1 18306.995,E2 18306.995} C_VEL
LIN {X 0,Y 423.035,Z 707.201,A -85,B 0,C 180,E1 18303.374,E2 18303.374} C_VEL
LIN {X 0,Y 426.82,Z 738.154,A -85,B 0,C 180,E1 18302.417,E2 18302.417} C_VEL
LIN {X 0,Y 423.104,Z 918.242,A -85,B 0,C 180,E1 18299.242,E2 18299.242} C_VEL
LIN {X 0,Y 422.016,Z 937.453,A -85,B 0,C 180,E1 18298.671,E2 18298.671} C_VEL
LIN {X 0,Y 420.651,Z 955.701,A -85,B 0,C 180,E1 18297.882,E2 18297.882} C_VEL
LIN {X 0,Y 419.065,Z 973.2,A -85,B 0,C 180,E1 18296.88,E2 18296.88} C_VEL
LIN {X 0,Y 417.322,Z 990.488,A -85,B 0,C 180,E1 18295.621,E2 18295.621} C_VEL
LIN {X 0,Y 415.496,Z 1007.262,A -85,B 0,C 180,E1 18294.106,E2 18294.106} C_VEL
LIN {X 0,Y 413.73,Z 1022.993,A -85,B 0,C 180,E1 18292.372,E2 18292.372} C_VEL
LIN {X 0,Y 412.147,Z 1037.488,A -85,B 0,C 180,E1 18290.447,E2 18290.447} C_VEL
LIN {X 0,Y 410.77,Z 1050.929,A -85,B 0,C 180,E1 18288.3,E2 18288.3} C_VEL
LIN {X 0,Y 409.707,Z 1063.1,A -85,B 0,C 180,E1 18285.945,E2 18285.945} C_VEL
LIN {X 0,Y 408.99,Z 1073.141,A -85,B 0,C 180,E1 18283.573,E2 18283.573} C_VEL
LIN {X 0,Y 408.591,Z 1081.584,A -85,B 0,C 180,E1 18281.103,E2 18281.103} C_VEL
LIN {X 0,Y 408.418,Z 1088.283,A -85,B 0,C 180,E1 18278.588,E2 18278.588} C_VEL
LIN {X 0,Y 408.405,Z 1093.247,A -85,B 0,C 180,E1 18276.043,E2 18276.043} C_VEL
LIN {X 0,Y 408.471,Z 1096.459,A -85,B 0,C 180,E1 18273.508,E2 18273.508} C_VEL
LIN {X 0,Y 408.518,Z 1097.982,A -85,B 0,C 180,E1 18270.981,E2 18270.981} C_VEL
LIN {X 0,Y 408.505,Z 1097.908,A -85,B 0,C 180,E1 18268.597,E2 18268.597} C_VEL
LIN {X 0,Y 408.442,Z 1096.166,A -85,B 0,C 180,E1 18266.069,E2 18266.069} C_VEL
LIN {X 0,Y 408.378,Z 1092.705,A -85,B 0,C 180,E1 18263.533,E2 18263.533} C_VEL
LIN {X 0,Y 408.413,Z 1087.479,A -85,B 0,C 180,E1 18260.985,E2 18260.985} C_VEL
LIN {X 0,Y 408.629,Z 1080.378,A -85,B 0,C 180,E1 18258.425,E2 18258.425} C_VEL
LIN {X 0,Y 409.087,Z 1071.768,A -85,B 0,C 180,E1 18255.997,E2 18255.997} C_VEL
LIN {X 0,Y 409.837,Z 1061.732,A -85,B 0,C 180,E1 18253.706,E2 18253.706} C_VEL
LIN {X 0,Y 410.94,Z 1049.535,A -85,B 0,C 180,E1 18251.413,E2 18251.413} C_VEL
LIN {X 0,Y 412.374,Z 1035.696,A -85,B 0,C 180,E1 18249.268,E2 18249.268} C_VEL
LIN {X 0,Y 414.003,Z 1020.626,A -85,B 0,C 180,E1 18247.343,E2 18247.343} C_VEL
LIN {X 0,Y 415.688,Z 1005.206,A -85,B 0,C 180,E1 18245.713,E2 18245.713} C_VEL
LIN {X 0,Y 417.389,Z 988.979,A -85,B 0,C 180,E1 18244.304,E2 18244.304} C_VEL
LIN {X 0,Y 419.008,Z 972.073,A -85,B 0,C 180,E1 18243.115,E2 18243.115} C_VEL
LIN {X 0,Y 420.559,Z 953.764,A -85,B 0,C 180,E1 18242.11,E2 18242.11} C_VEL
LIN {X 0,Y 421.861,Z 934.756,A -85,B 0,C 180,E1 18241.342,E2 18241.342} C_VEL
LIN {X 0,Y 422.785,Z 915.476,A -85,B 0,C 180,E1 18240.82,E2 18240.82} C_VEL
LIN {X 0,Y 425.917,Z 736.028,A -85,B 0,C 180,E1 18237.722,E2 18237.722} C_VEL
LIN {X 0,Y 422.24,Z 707.417,A -85,B 0,C 180,E1 18236.911,E2 18236.911} C_VEL
LIN {X 0,Y 425.897,Z 670.085,A -85,B 0,C 180,E1 18233.226,E2 18233.226} C_VEL
LIN {X 0,Y 419.446,Z 650.879,A -85,B 0,C 180,E1 18230.564,E2 18230.564} C_VEL
LIN {X 0,Y 412.378,Z 631.506,A -85,B 0,C 180,E1 18227.62,E2 18227.62} C_VEL
LIN {X 0,Y 409.466,Z 623.425,A -85,B 0,C 180,E1 18226.268,E2 18226.268} C_VEL
LIN {X 0,Y 409.435,Z 623.234,A -85,B 0,C 180,E1 18222.377,E2 18222.377} C_VEL
LIN {X 0,Y 409.433,Z 623.229,A -85,B 0,C 180,E1 18218.515,E2 18218.515} C_VEL
LIN {X 0,Y 409.436,Z 623.234,A -85,B 0,C 180,E1 18214.51,E2 18214.51} C_VEL
LIN {X 0,Y 409.445,Z 623.234,A -85,B 0,C 180,E1 18210.526,E2 18210.526} C_VEL
LIN {X 0,Y 409.442,Z 623.236,A -85,B 0,C 180,E1 18206.648,E2 18206.648} C_VEL
LIN {X 0,Y 409.445,Z 623.233,A -85,B 0,C 180,E1 18202.695,E2 18202.695} C_VEL
LIN {X 0,Y 409.439,Z 623.234,A -85,B 0,C 180,E1 18198.805,E2 18198.805} C_VEL
LIN {X 0,Y 409.413,Z 623.24,A -85,B 0,C 180,E1 18195.003,E2 18195.003} C_VEL
LIN {X 0,Y 409.446,Z 623.479,A -85,B 0,C 180,E1 18193.774,E2 18193.774} C_VEL
LIN {X 0,Y 413.844,Z 634.887,A -85,B 0,C 180,E1 18191.903,E2 18191.903} C_VEL
LIN {X 0,Y 418.177,Z 647.893,A -85,B 0,C 180,E1 18189.904,E2 18189.904} C_VEL
LIN {X 0,Y 420.836,Z 658.974,A -85,B 0,C 180,E1 18188.333,E2 18188.333} C_VEL
LIN {X 0,Y 420.275,Z 690.027,A -85,B 0,C 180,E1 18184.708,E2 18184.708} C_VEL
LIN {X 0,Y 419.683,Z 719.092,A -85,B 0,C 180,E1 18181.262,E2 18181.262} C_VEL
LIN {X 0,Y 419.873,Z 723.317,A -85,B 0,C 180,E1 18181.147,E2 18181.147} C_VEL
LIN {X 0,Y 416.955,Z 848.888,A -85,B 0,C 180,E1 18178.6,E2 18178.6} C_VEL
LIN {X 0,Y 416.875,Z 866.125,A -85,B 0,C 180,E1 18178.118,E2 18178.118} C_VEL
LIN {X 0,Y 416.478,Z 882.396,A -85,B 0,C 180,E1 18177.385,E2 18177.385} C_VEL
LIN {X 0,Y 415.888,Z 896.869,A -85,B 0,C 180,E1 18176.485,E2 18176.485} C_VEL
LIN {X 0,Y 415.055,Z 911.252,A -85,B 0,C 180,E1 18175.302,E2 18175.302} C_VEL
LIN {X 0,Y 414.204,Z 923.629,A -85,B 0,C 180,E1 18174.014,E2 18174.014} C_VEL
LIN {X 0,Y 413.235,Z 935.292,A -85,B 0,C 180,E1 18172.492,E2 18172.492} C_VEL
LIN {X 0,Y 412.287,Z 945.896,A -85,B 0,C 180,E1 18170.767,E2 18170.767} C_VEL
LIN {X 0,Y 411.429,Z 954.758,A -85,B 0,C 180,E1 18168.931,E2 18168.931} C_VEL
LIN {X 0,Y 410.689,Z 962.508,A -85,B 0,C 180,E1 18166.867,E2 18166.867} C_VEL
LIN {X 0,Y 410.113,Z 968.354,A -85,B 0,C 180,E1 18164.733,E2 18164.733} C_VEL
LIN {X 0,Y 409.709,Z 972.511,A -85,B 0,C 180,E1 18162.532,E2 18162.532} C_VEL
LIN {X 0,Y 409.457,Z 974.817,A -85,B 0,C 180,E1 18160.306,E2 18160.306} C_VEL
LIN {X 0,Y 409.344,Z 975.423,A -85,B 0,C 180,E1 18158.055,E2 18158.055} C_VEL
LIN {X 0,Y 409.331,Z 974.178,A -85,B 0,C 180,E1 18155.772,E2 18155.772} C_VEL
LIN {X 0,Y 409.457,Z 971.09,A -85,B 0,C 180,E1 18153.457,E2 18153.457} C_VEL
LIN {X 0,Y 409.74,Z 966.04,A -85,B 0,C 180,E1 18151.17,E2 18151.17} C_VEL
LIN {X 0,Y 410.181,Z 959.43,A -85,B 0,C 180,E1 18149.047,E2 18149.047} C_VEL
LIN {X 0,Y 410.798,Z 950.829,A -85,B 0,C 180,E1 18146.961,E2 18146.961} C_VEL
LIN {X 0,Y 411.507,Z 941.463,A -85,B 0,C 180,E1 18145.18,E2 18145.18} C_VEL
LIN {X 0,Y 412.407,Z 929.518,A -85,B 0,C 180,E1 18143.37,E2 18143.37} C_VEL
LIN {X 0,Y 413.295,Z 916.739,A -85,B 0,C 180,E1 18141.837,E2 18141.837} C_VEL
LIN {X 0,Y 414.166,Z 902.443,A -85,B 0,C 180,E1 18140.475,E2 18140.475} C_VEL
LIN {X 0,Y 414.939,Z 886.762,A -85,B 0,C 180,E1 18139.33,E2 18139.33} C_VEL
LIN {X 0,Y 415.507,Z 871.111,A -85,B 0,C 180,E1 18138.482,E2 18138.482} C_VEL
LIN {X 0,Y 415.854,Z 853.843,A -85,B 0,C 180,E1 18137.839,E2 18137.839} C_VEL
LIN {X 0,Y 416.143,Z 823.311,A -85,B 0,C 180,E1 18137.212,E2 18137.212} C_VEL
LIN {X 0,Y 418.037,Z 717.549,A -85,B 0,C 180,E1 18135.186,E2 18135.186} C_VEL
LIN {X 0,Y 416.693,Z 710.093,A -85,B 0,C 180,E1 18134.939,E2 18134.939} C_VEL
LIN {X 0,Y 417.624,Z 679.68,A -85,B 0,C 180,E1 18131.178,E2 18131.178} C_VEL
LIN {X 0,Y 418.179,Z 654.751,A -85,B 0,C 180,E1 18128.089,E2 18128.089} C_VEL
LIN {X 0,Y 413.424,Z 636.818,A -85,B 0,C 180,E1 18125.482,E2 18125.482} C_VEL
LIN {X 0,Y 411.155,Z 629.319,A -85,B 0,C 180,E1 18124.363,E2 18124.363} C_VEL
LIN {X 0,Y 409.229,Z 626.575,A -85,B 0,C 180,E1 18123.791,E2 18123.791} C_VEL
LIN {X 0,Y 405.701,Z 624.808,A -85,B 0,C 180,E1 18122.989,E2 18122.989} C_VEL
LIN {X 0,Y 402.298,Z 624.252,A -85,B 0,C 180,E1 18121.999,E2 18121.999} C_VEL
LIN {X 0,Y 401.489,Z 624.225,A -85,B 0,C 180,E1 18121.35,E2 18121.35} C_VEL
LIN {X 0,Y 401.497,Z 624.224,A -85,B 0,C 180,E1 18117.433,E2 18117.433} C_VEL
LIN {X 0,Y 401.481,Z 624.193,A -85,B 0,C 180,E1 18113.483,E2 18113.483} C_VEL
LIN {X 0,Y 401.501,Z 624.482,A -85,B 0,C 180,E1 18110.462,E2 18110.462} C_VEL
LIN {X 0,Y 406.429,Z 640.656,A -85,B 0,C 180,E1 18107.171,E2 18107.171} C_VEL
LIN {X 0,Y 411.059,Z 657.73,A -85,B 0,C 180,E1 18103.935,E2 18103.935} C_VEL
LIN {X 0,Y 412.158,Z 662.608,A -85,B 0,C 180,E1 18103.039,E2 18103.039} C_VEL
LIN {X 0,Y 409.552,Z 691.065,A -85,B 0,C 180,E1 18098.706,E2 18098.706} C_VEL
LIN {X 0,Y 409.253,Z 694.959,A -85,B 0,C 180,E1 18098.147,E2 18098.147} C_VEL
LIN {X 0,Y 414.665,Z 722.892,A -85,B 0,C 180,E1 18097.211,E2 18097.211} C_VEL
LIN {X 0,Y 412.308,Z 845.992,A -85,B 0,C 180,E1 18094.983,E2 18094.983} C_VEL
LIN {X 0,Y 411.748,Z 863.164,A -85,B 0,C 180,E1 18094.4,E2 18094.4} C_VEL
